LIN {X 0,Y 191.583,Z 536.213,A -85,B 0,C 180,E1 -22027.347,E2 -22027.347} C_VEL
LIN {X 0,Y 188.784,Z 540.752,A -85,B 0,C 180,E1 -22030.427,E2 -22030.427} C_VEL
LIN {X 0,Y 187.171,Z 543.158,A -85,B 0,C 180,E1 -22032.521,E2 -22032.521} C_VEL
LIN {X 0,Y 184.868,Z 546.72,A -85,B 0,C 180,E1 -22036.817,E2 -22036.817} C_VEL
LIN {X 0,Y 184.098,Z 547.887,A -85,B 0,C 180,E1 -22038.998,E2 -22038.998} C_VEL
LIN {X 0,Y 183.22,Z 549.005,A -85,B 0,C 180,E1 -22043.394,E2 -22043.394} C_VEL
LIN {X 0,Y 183.101,Z 548.604,A -85,B 0,C 180,E1 -22047.802,E2 -22047.802} C_VEL
LIN {X 0,Y 183.237,Z 547.778,A -85,B 0,C 180,E1 -22050.002,E2 -22050.002} C_VEL
LIN {X 0,Y 183.088,Z 545.543,A -85,B 0,C 180,E1 -22053.583,E2 -22053.583} C_VEL
LIN {X 0,Y 183.262,Z 542.775,A -85,B 0,C 180,E1 -22056.608,E2 -22056.608} C_VEL
LIN {X 0,Y 183.704,Z 538.696,A -85,B 0,C 180,E1 -22059.915,E2 -22059.915} C_VEL
LIN {X 0,Y 184.708,Z 532.396,A -85,B 0,C 180,E1 -22063.759,E2 -22063.759} C_VEL
LIN {X 0,Y 186.239,Z 525.529,A -85,B 0,C 180,E1 -22067.007,E2 -22067.007} C_VEL
LIN {X 0,Y 187.918,Z 518.509,A -85,B 0,C 180,E1 -22069.671,E2 -22069.671} C_VEL
LIN {X 0,Y 189.702,Z 510.19,A -85,B 0,C 180,E1 -22072.261,E2 -22072.261} C_VEL
LIN {X 0,Y 191.808,Z 500.693,A -85,B 0,C 180,E1 -22074.634,E2 -22074.634} C_VEL
LIN {X 0,Y 194.283,Z 489.109,A -85,B 0,C 180,E1 -22076.885,E2 -22076.885} C_VEL
LIN {X 0,Y 196.502,Z 477.732,A -85,B 0,C 180,E1 -22078.581,E2 -22078.581} C_VEL
LIN {X 0,Y 198.278,Z 466.082,A -85,B 0,C 180,E1 -22079.899,E2 -22079.899} C_VEL
LIN {X 0,Y 199.683,Z 453.556,A -85,B 0,C 180,E1 -22080.908,E2 -22080.908} C_VEL
LIN {X 0,Y 200.634,Z 440.994,A -85,B 0,C 180,E1 -22081.552,E2 -22081.552} C_VEL
LIN {X 0,Y 202.544,Z 391.87,A -85,B 0,C 180,E1 -22083.238,E2 -22083.238} C_VEL
LIN {X 0,Y 200.132,Z 369.782,A -85,B 0,C 180,E1 -22084.491,E2 -22084.491} C_VEL
LIN {X 0,Y 194.209,Z 353.858,A -85,B 0,C 180,E1 -22086.126,E2 -22086.126} C_VEL
LIN {X 0,Y 188.089,Z 340.011,A -85,B 0,C 180,E1 -22087.833,E2 -22087.833} C_VEL
LIN {X 0,Y 186.441,Z 336.416,A -85,B 0,C 180,E1 -22088.331,E2 -22088.331} C_VEL
LIN {X 0,Y 185.481,Z 332.385,A -85,B 0,C 180,E1 -22090.619,E2 -22090.619} C_VEL
LIN {X 0,Y 185.463,Z 332.386,A -85,B 0,C 180,E1 -22096.056,E2 -22096.056} C_VEL
LIN {X 0,Y 185.473,Z 332.384,A -85,B 0,C 180,E1 -22099.896,E2 -22099.896} C_VEL
LIN {X 0,Y 185.512,Z 332.378,A -85,B 0,C 180,E1 -22102.712,E2 -22102.712} C_VEL
LIN {X 0,Y 185.536,Z 332.372,A -85,B 0,C 180,E1 -22107.973,E2 -22107.973} C_VEL
LIN {X 0,Y 185.553,Z 332.371,A -85,B 0,C 180,E1 -22110.596,E2 -22110.596} C_VEL
LIN {X 0,Y 185.586,Z 332.368,A -85,B 0,C 180,E1 -22115.382,E2 -22115.382} C_VEL
LIN {X 0,Y 185.634,Z 332.342,A -85,B 0,C 180,E1 -22121.176,E2 -22121.176} C_VEL
LIN {X 0,Y 185.676,Z 332.354,A -85,B 0,C 180,E1 -22124.635,E2 -22124.635} C_VEL
LIN {X 0,Y 185.894,Z 332.304,A -85,B 0,C 180,E1 -22129.418,E2 -22129.418} C_VEL
LIN {X 0,Y 185.943,Z 332.31,A -85,B 0,C 180,E1 -22133.489,E2 -22133.489} C_VEL
LIN {X 0,Y 186.187,Z 332.289,A -85,B 0,C 180,E1 -22137.836,E2 -22137.836} C_VEL
LIN {X 0,Y 186.402,Z 332.248,A -85,B 0,C 180,E1 -22139.999,E2 -22139.999} C_VEL
LIN {X 0,Y 185.898,Z 332.304,A -85,B 0,C 180,E1 -22144.336,E2 -22144.336} C_VEL
LIN {X 0,Y 185.981,Z 332.318,A -85,B 0,C 180,E1 -22148.693,E2 -22148.693} C_VEL
LIN {X 0,Y 185.724,Z 332.33,A -85,B 0,C 180,E1 -22153.123,E2 -22153.123} C_VEL
LIN {X 0,Y 185.659,Z 332.34,A -85,B 0,C 180,E1 -22157.627,E2 -22157.627} C_VEL
LIN {X 0,Y 185.571,Z 332.367,A -85,B 0,C 180,E1 -22162.254,E2 -22162.254} C_VEL
LIN {X 0,Y 185.582,Z 332.355,A -85,B 0,C 180,E1 -22164.645,E2 -22164.645} C_VEL
LIN {X 0,Y 185.548,Z 332.348,A -85,B 0,C 180,E1 -22169.498,E2 -22169.498} C_VEL
LIN {X 0,Y 185.501,Z 332.372,A -85,B 0,C 180,E1 -22174.631,E2 -22174.631} C_VEL
LIN {X 0,Y 185.508,Z 332.351,A -85,B 0,C 180,E1 -22177.312,E2 -22177.312} C_VEL
LIN {X 0,Y 185.474,Z 332.369,A -85,B 0,C 180,E1 -22180.723,E2 -22180.723} C_VEL
LIN {X 0,Y 185.461,Z 332.368,A -85,B 0,C 180,E1 -22186.054,E2 -22186.054} C_VEL
LIN {X 0,Y 185.47,Z 332.375,A -85,B 0,C 180,E1 -22189.894,E2 -22189.894} C_VEL
LIN {X 0,Y 185.509,Z 332.374,A -85,B 0,C 180,E1 -22192.71,E2 -22192.71} C_VEL
LIN {X 0,Y 185.533,Z 332.374,A -85,B 0,C 180,E1 -22197.971,E2 -22197.971} C_VEL
LIN {X 0,Y 185.549,Z 332.373,A -85,B 0,C 180,E1 -22200.593,E2 -22200.593} C_VEL
LIN {X 0,Y 185.612,Z 332.364,A -85,B 0,C 180,E1 -22205.789,E2 -22205.789} C_VEL
LIN {X 0,Y 186.61,Z 335.177,A -85,B 0,C 180,E1 -22206.126,E2 -22206.126} C_VEL
LIN {X 0,Y 188.138,Z 337.771,A -85,B 0,C 180,E1 -22206.537,E2 -22206.537} C_VEL
LIN {X 0,Y 195.669,Z 351.908,A -85,B 0,C 180,E1 -22208.504,E2 -22208.504} C_VEL
LIN {X 0,Y 199.025,Z 359.752,A -85,B 0,C 180,E1 -22209.387,E2 -22209.387} C_VEL
LIN {X 0,Y 203.412,Z 372.384,A -85,B 0,C 180,E1 -22210.581,E2 -22210.581} C_VEL
LIN {X 0,Y 200.56,Z 435.216,A -85,B 0,C 180,E1 -22212.716,E2 -22212.716} C_VEL
LIN {X 0,Y 199.337,Z 448.756,A -85,B 0,C 180,E1 -22213.562,E2 -22213.562} C_VEL
LIN {X 0,Y 197.947,Z 460.625,A -85,B 0,C 180,E1 -22214.687,E2 -22214.687} C_VEL
LIN {X 0,Y 196.128,Z 472.793,A -85,B 0,C 180,E1 -22216.265,E2 -22216.265} C_VEL
LIN {X 0,Y 193.844,Z 484.802,A -85,B 0,C 180,E1 -22218.321,E2 -22218.321} C_VEL
LIN {X 0,Y 191.638,Z 494.794,A -85,B 0,C 180,E1 -22220.499,E2 -22220.499} C_VEL
LIN {X 0,Y 189.47,Z 504.15,A -85,B 0,C 180,E1 -22223.074,E2 -22223.074} C_VEL
LIN {X 0,Y 187.292,Z 513.207,A -85,B 0,C 180,E1 -22226.233,E2 -22226.233} C_VEL
LIN {X 0,Y 185.605,Z 520.503,A -85,B 0,C 180,E1 -22229.456,E2 -22229.456} C_VEL
LIN {X 0,Y 184.53,Z 525.43,A -85,B 0,C 180,E1 -22232.181,E2 -22232.181} C_VEL
LIN {X 0,Y 183.676,Z 530.659,A -85,B 0,C 180,E1 -22235.83,E2 -22235.83} C_VEL
LIN {X 0,Y 183.13,Z 533.887,A -85,B 0,C 180,E1 -22238.828,E2 -22238.828} C_VEL
LIN {X 0,Y 182.842,Z 535.784,A -85,B 0,C 180,E1 -22241.078,E2 -22241.078} C_VEL
LIN {X 0,Y 182.796,Z 537.198,A -85,B 0,C 180,E1 -22243.335,E2 -22243.335} C_VEL
LIN {X 0,Y 182.939,Z 538.419,A -85,B 0,C 180,E1 -22246.174,E2 -22246.174} C_VEL
LIN {X 0,Y 183.416,Z 538.99,A -85,B 0,C 180,E1 -22250.171,E2 -22250.171} C_VEL
LIN {X 0,Y 184.48,Z 538.359,A -85,B 0,C 180,E1 -22253.893,E2 -22253.893} C_VEL
LIN {X 0,Y 185.784,Z 536.971,A -85,B 0,C 180,E1 -22256.995,E2 -22256.995} C_VEL
LIN {X 0,Y 187.959,Z 534.14,A -85,B 0,C 180,E1 -22260.685,E2 -22260.685} C_VEL
LIN {X 0,Y 191.223,Z 529.402,A -85,B 0,C 180,E1 -22264.725,E2 -22264.725} C_VEL
LIN {X 0,Y 195.104,Z 523.18,A -85,B 0,C 180,E1 -22268.414,E2 -22268.414} C_VEL
LIN {X 0,Y 198.974,Z 516.267,A -85,B 0,C 180,E1 -22271.471,E2 -22271.471} C_VEL
LIN {X 0,Y 202.688,Z 509.169,A -85,B 0,C 180,E1 -22273.903,E2 -22273.903} C_VEL
LIN {X 0,Y 206.691,Z 500.537,A -85,B 0,C 180,E1 -22276.262,E2 -22276.262} C_VEL
LIN {X 0,Y 210.474,Z 491.374,A -85,B 0,C 180,E1 -22278.23,E2 -22278.23} C_VEL
LIN {X 0,Y 214.251,Z 480.505,A -85,B 0,C 180,E1 -22280.061,E2 -22280.061} C_VEL
LIN {X 0,Y 217.541,Z 469.264,A -85,B 0,C 180,E1 -22281.513,E2 -22281.513} C_VEL
LIN {X 0,Y 220.372,Z 457.031,A -85,B 0,C 180,E1 -22282.704,E2 -22282.704} C_VEL
LIN {X 0,Y 222.473,Z 443.681,A -85,B 0,C 180,E1 -22283.632,E2 -22283.632} C_VEL
LIN {X 0,Y 223.846,Z 430.846,A -85,B 0,C 180,E1 -22284.167,E2 -22284.167} C_VEL
LIN {X 0,Y 226.225,Z 394.156,A -85,B 0,C 180,E1 -22285.231,E2 -22285.231} C_VEL
LIN {X 0,Y 220.963,Z 383.068,A -85,B 0,C 180,E1 -22287.269,E2 -22287.269} C_VEL
LIN {X 0,Y 215.515,Z 372.798,A -85,B 0,C 180,E1 -22289.527,E2 -22289.527} C_VEL
LIN {X 0,Y 211.22,Z 365.794,A -85,B 0,C 180,E1 -22291.426,E2 -22291.426} C_VEL
LIN {X 0,Y 205.505,Z 357.753,A -85,B 0,C 180,E1 -22294.149,E2 -22294.149} C_VEL
LIN {X 0,Y 201.846,Z 352.98,A -85,B 0,C 180,E1 -22296.063,E2 -22296.063} C_VEL
LIN {X 0,Y 199.159,Z 349.322,A -85,B 0,C 180,E1 -22297.596,E2 -22297.596} C_VEL
LIN {X 0,Y 195.776,Z 345.444,A -85,B 0,C 180,E1 -22299.658,E2 -22299.658} C_VEL
LIN {X 0,Y 194.816,Z 343.709,A -85,B 0,C 180,E1 -22300.336,E2 -22300.336} C_VEL
LIN {X 0,Y 192.254,Z 341.564,A -85,B 0,C 180,E1 -22302.047,E2 -22302.047} C_VEL
LIN {X 0,Y 190.274,Z 338.16,A -85,B 0,C 180,E1 -22303.642,E2 -22303.642} C_VEL
LIN {X 0,Y 187.582,Z 336.397,A -85,B 0,C 180,E1 -22305.767,E2 -22305.767} C_VEL
LIN {X 0,Y 186.189,Z 334.174,A -85,B 0,C 180,E1 -22307.119,E2 -22307.119} C_VEL
LIN {X 0,Y 185.73,Z 332.335,A -85,B 0,C 180,E1 -22307.78,E2 -22307.78} C_VEL
LIN {X 0,Y 185.963,Z 332.3,A -85,B 0,C 180,E1 -22311.306,E2 -22311.306} C_VEL
LIN {X 0,Y 186.148,Z 332.28,A -85,B 0,C 180,E1 -22317.837,E2 -22317.837} C_VEL
LIN {X 0,Y 186.366,Z 332.267,A -85,B 0,C 180,E1 -22320.001,E2 -22320.001} C_VEL
LIN {X 0,Y 185.873,Z 332.325,A -85,B 0,C 180,E1 -22324.337,E2 -22324.337} C_VEL
LIN {X 0,Y 185.967,Z 332.299,A -85,B 0,C 180,E1 -22328.695,E2 -22328.695} C_VEL
LIN {X 0,Y 185.714,Z 332.328,A -85,B 0,C 180,E1 -22333.125,E2 -22333.125} C_VEL
LIN {X 0,Y 185.677,Z 332.335,A -85,B 0,C 180,E1 -22337.627,E2 -22337.627} C_VEL
LIN {X 0,Y 185.605,Z 332.347,A -85,B 0,C 180,E1 -22343.428,E2 -22343.428} C_VEL
LIN {X 0,Y 185.596,Z 332.595,A -85,B 0,C 180,E1 -22344.664,E2 -22344.664} C_VEL
LIN {X 0,Y 185.914,Z 333.985,A -85,B 0,C 180,E1 -22346.295,E2 -22346.295} C_VEL
LIN {X 0,Y 187.303,Z 336.241,A -85,B 0,C 180,E1 -22347.668,E2 -22347.668} C_VEL
LIN {X 0,Y 191.692,Z 341.119,A -85,B 0,C 180,E1 -22351.222,E2 -22351.222} C_VEL
LIN {X 0,Y 195.213,Z 346.119,A -85,B 0,C 180,E1 -22353.745,E2 -22353.745} C_VEL
LIN {X 0,Y 196.675,Z 348.072,A -85,B 0,C 180,E1 -22354.698,E2 -22354.698} C_VEL
LIN {X 0,Y 200.777,Z 353.997,A -85,B 0,C 180,E1 -22357.174,E2 -22357.174} C_VEL
LIN {X 0,Y 204.53,Z 359.728,A -85,B 0,C 180,E1 -22359.228,E2 -22359.228} C_VEL
LIN {X 0,Y 208.687,Z 366.484,A -85,B 0,C 180,E1 -22361.325,E2 -22361.325} C_VEL
LIN {X 0,Y 213.965,Z 375.728,A -85,B 0,C 180,E1 -22363.769,E2 -22363.769} C_VEL
LIN {X 0,Y 218.853,Z 385.288,A -85,B 0,C 180,E1 -22365.862,E2 -22365.862} C_VEL
LIN {X 0,Y 224.441,Z 397.981,A -85,B 0,C 180,E1 -22368.12,E2 -22368.12} C_VEL
LIN {X 0,Y 225.844,Z 401.455,A -85,B 0,C 180,E1 -22368.668,E2 -22368.668} C_VEL
LIN {X 0,Y 222.983,Z 445.282,A -85,B 0,C 180,E1 -22370.003,E2 -22370.003} C_VEL
LIN {X 0,Y 222.619,Z 448.507,A -85,B 0,C 180,E1 -22370.137,E2 -22370.137} C_VEL
LIN {X 0,Y 221.356,Z 454.274,A -85,B 0,C 180,E1 -22370.283,E2 -22370.283} C_VEL
LIN {X 0,Y 217.615,Z 463.501,A -85,B 0,C 180,E1 -22370.319,E2 -22370.319} C_VEL
LIN {X 0,Y 213.48,Z 472.458,A -85,B 0,C 180,E1 -22370.543,E2 -22370.543} C_VEL
LIN {X 0,Y 211.606,Z 477.79,A -85,B 0,C 180,E1 -22370.988,E2 -22370.988} C_VEL
LIN {X 0,Y 207.869,Z 489.719,A -85,B 0,C 180,E1 -22372.516,E2 -22372.516} C_VEL
LIN {X 0,Y 203.592,Z 500.823,A -85,B 0,C 180,E1 -22374.374,E2 -22374.374} C_VEL
LIN {X 0,Y 199.718,Z 509.796,A -85,B 0,C 180,E1 -22376.344,E2 -22376.344} C_VEL
LIN {X 0,Y 194.763,Z 519.539,A -85,B 0,C 180,E1 -22379.058,E2 -22379.058} C_VEL
LIN {X 0,Y 190.378,Z 527.383,A -85,B 0,C 180,E1 -22381.924,E2 -22381.924} C_VEL
LIN {X 0,Y 186.832,Z 533.565,A -85,B 0,C 180,E1 -22384.897,E2 -22384.897} C_VEL
LIN {X 0,Y 183.033,Z 539.419,A -85,B 0,C 180,E1 -22388.609,E2 -22388.609} C_VEL
LIN {X 0,Y 180.412,Z 543.169,A -85,B 0,C 180,E1 -22391.844,E2 -22391.844} C_VEL
LIN {X 0,Y 178.996,Z 545.117,A -85,B 0,C 180,E1 -22394.05,E2 -22394.05} C_VEL
LIN {X 0,Y 177.945,Z 546.661,A -85,B 0,C 180,E1 -22396.294,E2 -22396.294} C_VEL
LIN {X 0,Y 176.509,Z 548.482,A -85,B 0,C 180,E1 -22400.838,E2 -22400.838} C_VEL
LIN {X 0,Y 176.008,Z 548.783,A -85,B 0,C 180,E1 -22405.422,E2 -22405.422} C_VEL
LIN {X 0,Y 176.019,Z 548.334,A -85,B 0,C 180,E1 -22407.714,E2 -22407.714} C_VEL
LIN {X 0,Y 176.141,Z 547.469,A -85,B 0,C 180,E1 -22410.002,E2 -22410.002} C_VEL
LIN {X 0,Y 175.997,Z 545.487,A -85,B 0,C 180,E1 -22413.321,E2 -22413.321} C_VEL
LIN {X 0,Y 176.205,Z 542.333,A -85,B 0,C 180,E1 -22416.874,E2 -22416.874} C_VEL
LIN {X 0,Y 176.671,Z 538.178,A -85,B 0,C 180,E1 -22420.314,E2 -22420.314} C_VEL
LIN {X 0,Y 177.759,Z 531.795,A -85,B 0,C 180,E1 -22424.308,E2 -22424.308} C_VEL
LIN {X 0,Y 179.431,Z 524.841,A -85,B 0,C 180,E1 -22427.673,E2 -22427.673} C_VEL
LIN {X 0,Y 181.234,Z 517.72,A -85,B 0,C 180,E1 -22430.429,E2 -22430.429} C_VEL
LIN {X 0,Y 183.18,Z 509.067,A -85,B 0,C 180,E1 -22433.159,E2 -22433.159} C_VEL
LIN {X 0,Y 185.676,Z 498.382,A -85,B 0,C 180,E1 -22435.805,E2 -22435.805} C_VEL
LIN {X 0,Y 187.629,Z 489.212,A -85,B 0,C 180,E1 -22437.617,E2 -22437.617} C_VEL
LIN {X 0,Y 189.926,Z 477.908,A -85,B 0,C 180,E1 -22439.362,E2 -22439.362} C_VEL
LIN {X 0,Y 191.766,Z 466.4,A -85,B 0,C 180,E1 -22440.719,E2 -22440.719} C_VEL
LIN {X 0,Y 193.327,Z 453.215,A -85,B 0,C 180,E1 -22441.813,E2 -22441.813} C_VEL
LIN {X 0,Y 194.305,Z 440.553,A -85,B 0,C 180,E1 -22442.475,E2 -22442.475} C_VEL
LIN {X 0,Y 196.253,Z 392.537,A -85,B 0,C 180,E1 -22444.167,E2 -22444.167} C_VEL
LIN {X 0,Y 194.04,Z 371.837,A -85,B 0,C 180,E1 -22445.392,E2 -22445.392} C_VEL
LIN {X 0,Y 187.655,Z 354.77,A -85,B 0,C 180,E1 -22447.26,E2 -22447.26} C_VEL
LIN {X 0,Y 182.372,Z 343.133,A -85,B 0,C 180,E1 -22448.812,E2 -22448.812} C_VEL
LIN {X 0,Y 179.102,Z 336.151,A -85,B 0,C 180,E1 -22449.857,E2 -22449.857} C_VEL
LIN {X 0,Y 178.406,Z 333.266,A -85,B 0,C 180,E1 -22451.695,E2 -22451.695} C_VEL
LIN {X 0,Y 178.397,Z 333.268,A -85,B 0,C 180,E1 -22455.165,E2 -22455.165} C_VEL
LIN {X 0,Y 178.408,Z 333.263,A -85,B 0,C 180,E1 -22458.46,E2 -22458.46} C_VEL
LIN {X 0,Y 178.428,Z 333.26,A -85,B 0,C 180,E1 -22463.784,E2 -22463.784} C_VEL
LIN {X 0,Y 178.489,Z 333.251,A -85,B 0,C 180,E1 -22466.547,E2 -22466.547} C_VEL
LIN {X 0,Y 178.45,Z 333.254,A -85,B 0,C 180,E1 -22471.796,E2 -22471.796} C_VEL
LIN {X 0,Y 178.521,Z 333.247,A -85,B 0,C 180,E1 -22474.889,E2 -22474.889} C_VEL
LIN {X 0,Y 178.563,Z 333.22,A -85,B 0,C 180,E1 -22480.845,E2 -22480.845} C_VEL
LIN {X 0,Y 178.651,Z 333.228,A -85,B 0,C 180,E1 -22486.347,E2 -22486.347} C_VEL
LIN {X 0,Y 178.913,Z 333.167,A -85,B 0,C 180,E1 -22490.959,E2 -22490.959} C_VEL
LIN {X 0,Y 178.849,Z 333.203,A -85,B 0,C 180,E1 -22495.492,E2 -22495.492} C_VEL
LIN {X 0,Y 179.366,Z 333.124,A -85,B 0,C 180,E1 -22499.999,E2 -22499.999} C_VEL
LIN {X 0,Y 178.904,Z 333.194,A -85,B 0,C 180,E1 -22506.768,E2 -22506.768} C_VEL
LIN {X 0,Y 178.838,Z 333.202,A -85,B 0,C 180,E1 -22510.741,E2 -22510.741} C_VEL
LIN {X 0,Y 178.595,Z 333.204,A -85,B 0,C 180,E1 -22515.989,E2 -22515.989} C_VEL
LIN {X 0,Y 178.561,Z 333.234,A -85,B 0,C 180,E1 -22519.153,E2 -22519.153} C_VEL
LIN {X 0,Y 178.52,Z 333.229,A -85,B 0,C 180,E1 -22525.11,E2 -22525.11} C_VEL
LIN {X 0,Y 178.464,Z 333.241,A -85,B 0,C 180,E1 -22530.793,E2 -22530.793} C_VEL
LIN {X 0,Y 178.487,Z 333.245,A -85,B 0,C 180,E1 -22534.217,E2 -22534.217} C_VEL
LIN {X 0,Y 178.398,Z 333.233,A -85,B 0,C 180,E1 -22539.073,E2 -22539.073} C_VEL
LIN {X 0,Y 178.401,Z 333.257,A -85,B 0,C 180,E1 -22542.044,E2 -22542.044} C_VEL
LIN {X 0,Y 178.396,Z 333.255,A -85,B 0,C 180,E1 -22545.163,E2 -22545.163} C_VEL
LIN {X 0,Y 178.405,Z 333.243,A -85,B 0,C 180,E1 -22548.458,E2 -22548.458} C_VEL
LIN {X 0,Y 178.424,Z 333.249,A -85,B 0,C 180,E1 -22553.781,E2 -22553.781} C_VEL
LIN {X 0,Y 178.486,Z 333.243,A -85,B 0,C 180,E1 -22556.544,E2 -22556.544} C_VEL
LIN {X 0,Y 178.446,Z 333.256,A -85,B 0,C 180,E1 -22561.794,E2 -22561.794} C_VEL
LIN {X 0,Y 178.496,Z 333.353,A -85,B 0,C 180,E1 -22564.373,E2 -22564.373} C_VEL
LIN {X 0,Y 179.446,Z 336.032,A -85,B 0,C 180,E1 -22564.706,E2 -22564.706} C_VEL
LIN {X 0,Y 181.005,Z 338.354,A -85,B 0,C 180,E1 -22565.145,E2 -22565.145} C_VEL
LIN {X 0,Y 188.936,Z 353.033,A -85,B 0,C 180,E1 -22567.362,E2 -22567.362} C_VEL
LIN {X 0,Y 192.65,Z 361.062,A -85,B 0,C 180,E1 -22568.375,E2 -22568.375} C_VEL
LIN {X 0,Y 197.1,Z 373.943,A -85,B 0,C 180,E1 -22569.662,E2 -22569.662} C_VEL
LIN {X 0,Y 194.252,Z 434.941,A -85,B 0,C 180,E1 -22571.786,E2 -22571.786} C_VEL
LIN {X 0,Y 193.019,Z 448.221,A -85,B 0,C 180,E1 -22572.62,E2 -22572.62} C_VEL
LIN {X 0,Y 191.58,Z 460.11,A -85,B 0,C 180,E1 -22573.755,E2 -22573.755} C_VEL
LIN {X 0,Y 189.8,Z 471.658,A -85,B 0,C 180,E1 -22575.25,E2 -22575.25} C_VEL
LIN {X 0,Y 187.78,Z 482.209,A -85,B 0,C 180,E1 -22577.021,E2 -22577.021} C_VEL
LIN {X 0,Y 185.382,Z 493.034,A -85,B 0,C 180,E1 -22579.348,E2 -22579.348} C_VEL
LIN {X 0,Y 182.843,Z 503.663,A -85,B 0,C 180,E1 -22582.267,E2 -22582.267} C_VEL
LIN {X 0,Y 180.516,Z 512.847,A -85,B 0,C 180,E1 -22585.532,E2 -22585.532} C_VEL
LIN {X 0,Y 178.709,Z 520.242,A -85,B 0,C 180,E1 -22588.871,E2 -22588.871} C_VEL
LIN {X 0,Y 177.385,Z 526.17,A -85,B 0,C 180,E1 -22592.269,E2 -22592.269} C_VEL
LIN {X 0,Y 176.598,Z 530.93,A -85,B 0,C 180,E1 -22595.786,E2 -22595.786} C_VEL
LIN {X 0,Y 175.968,Z 534.411,A -85,B 0,C 180,E1 -22599.191,E2 -22599.191} C_VEL
LIN {X 0,Y 175.711,Z 536.209,A -85,B 0,C 180,E1 -22601.534,E2 -22601.534} C_VEL
LIN {X 0,Y 175.693,Z 537.573,A -85,B 0,C 180,E1 -22603.885,E2 -22603.885} C_VEL
LIN {X 0,Y 175.85,Z 538.601,A -85,B 0,C 180,E1 -22606.429,E2 -22606.429} C_VEL
LIN {X 0,Y 176.072,Z 539.077,A -85,B 0,C 180,E1 -22608.62,E2 -22608.62} C_VEL
LIN {X 0,Y 176.482,Z 539.171,A -85,B 0,C 180,E1 -22611,E2 -22611} C_VEL
LIN {X 0,Y 177.534,Z 538.59,A -85,B 0,C 180,E1 -22614.427,E2 -22614.427} C_VEL
LIN {X 0,Y 179.164,Z 536.952,A -85,B 0,C 180,E1 -22618.079,E2 -22618.079} C_VEL
LIN {X 0,Y 181.263,Z 534.421,A -85,B 0,C 180,E1 -22621.462,E2 -22621.462} C_VEL
LIN {X 0,Y 184.076,Z 530.632,A -85,B 0,C 180,E1 -22624.936,E2 -22624.936} C_VEL
LIN {X 0,Y 187.649,Z 525.405,A -85,B 0,C 180,E1 -22628.393,E2 -22628.393} C_VEL
LIN {X 0,Y 191.292,Z 519.43,A -85,B 0,C 180,E1 -22631.397,E2 -22631.397} C_VEL
LIN {X 0,Y 195.818,Z 511.415,A -85,B 0,C 180,E1 -22634.47,E2 -22634.47} C_VEL
LIN {X 0,Y 199.885,Z 503.351,A -85,B 0,C 180,E1 -22636.848,E2 -22636.848} C_VEL
LIN {X 0,Y 204.347,Z 493.283,A -85,B 0,C 180,E1 -22639.165,E2 -22639.165} C_VEL
LIN {X 0,Y 208.117,Z 483.339,A -85,B 0,C 180,E1 -22640.956,E2 -22640.956} C_VEL
LIN {X 0,Y 211.591,Z 472.542,A -85,B 0,C 180,E1 -22642.464,E2 -22642.464} C_VEL
LIN {X 0,Y 214.654,Z 460.43,A -85,B 0,C 180,E1 -22643.746,E2 -22643.746} C_VEL
LIN {X 0,Y 217.154,Z 446.95,A -85,B 0,C 180,E1 -22644.777,E2 -22644.777} C_VEL
LIN {X 0,Y 218.683,Z 434.418,A -85,B 0,C 180,E1 -22645.389,E2 -22645.389} C_VEL
LIN {X 0,Y 221.27,Z 396.686,A -85,B 0,C 180,E1 -22646.51,E2 -22646.51} C_VEL
LIN {X 0,Y 215.722,Z 385.017,A -85,B 0,C 180,E1 -22648.81,E2 -22648.81} C_VEL
LIN {X 0,Y 210.131,Z 374.508,A -85,B 0,C 180,E1 -22651.332,E2 -22651.332} C_VEL
LIN {X 0,Y 205.06,Z 366.991,A -85,B 0,C 180,E1 -22653.76,E2 -22653.76} C_VEL
LIN {X 0,Y 202.037,Z 362.773,A -85,B 0,C 180,E1 -22655.328,E2 -22655.328} C_VEL
LIN {X 0,Y 199.351,Z 359.105,A -85,B 0,C 180,E1 -22656.817,E2 -22656.817} C_VEL
LIN {X 0,Y 195.958,Z 354.595,A -85,B 0,C 180,E1 -22658.854,E2 -22658.854} C_VEL
LIN {X 0,Y 193.374,Z 351.4,A -85,B 0,C 180,E1 -22660.546,E2 -22660.546} C_VEL
LIN {X 0,Y 192.535,Z 350.125,A -85,B 0,C 180,E1 -22661.147,E2 -22661.147} C_VEL
LIN {X 0,Y 189.968,Z 347.519,A -85,B 0,C 180,E1 -22662.993,E2 -22662.993} C_VEL
LIN {X 0,Y 188.414,Z 344.857,A -85,B 0,C 180,E1 -22664.311,E2 -22664.311} C_VEL
LIN {X 0,Y 185.69,Z 342.747,A -85,B 0,C 180,E1 -22666.596,E2 -22666.596} C_VEL
LIN {X 0,Y 184.14,Z 339.969,A -85,B 0,C 180,E1 -22668.232,E2 -22668.232} C_VEL
LIN {X 0,Y 183.748,Z 339.136,A -85,B 0,C 180,E1 -22668.696,E2 -22668.696} C_VEL
LIN {X 0,Y 180.696,Z 337.123,A -85,B 0,C 180,E1 -22672.177,E2 -22672.177} C_VEL
LIN {X 0,Y 179.132,Z 334.564,A -85,B 0,C 180,E1 -22674.654,E2 -22674.654} C_VEL
LIN {X 0,Y 178.816,Z 333.195,A -85,B 0,C 180,E1 -22675.492,E2 -22675.492} C_VEL
LIN {X 0,Y 179.331,Z 333.142,A -85,B 0,C 180,E1 -22680.001,E2 -22680.001} C_VEL
LIN {X 0,Y 178.822,Z 333.205,A -85,B 0,C 180,E1 -22684.509,E2 -22684.509} C_VEL
LIN {X 0,Y 178.898,Z 333.182,A -85,B 0,C 180,E1 -22689.041,E2 -22689.041} C_VEL
LIN {X 0,Y 178.642,Z 333.209,A -85,B 0,C 180,E1 -22693.654,E2 -22693.654} C_VEL
LIN {X 0,Y 178.653,Z 333.346,A -85,B 0,C 180,E1 -22698.047,E2 -22698.047} C_VEL
LIN {X 0,Y 179.263,Z 335.526,A -85,B 0,C 180,E1 -22699.371,E2 -22699.371} C_VEL
LIN {X 0,Y 181,Z 337.81,A -85,B 0,C 180,E1 -22701.946,E2 -22701.946} C_VEL
LIN {X 0,Y 183.17,Z 339.266,A -85,B 0,C 180,E1 -22704.434,E2 -22704.434} C_VEL
LIN {X 0,Y 184.264,Z 340.742,A -85,B 0,C 180,E1 -22705.637,E2 -22705.637} C_VEL
LIN {X 0,Y 186.143,Z 343.345,A -85,B 0,C 180,E1 -22707.498,E2 -22707.498} C_VEL
LIN {X 0,Y 189.689,Z 347.557,A -85,B 0,C 180,E1 -22710.492,E2 -22710.492} C_VEL
LIN {X 0,Y 193.668,Z 353.099,A -85,B 0,C 180,E1 -22713.425,E2 -22713.425} C_VEL
LIN {X 0,Y 198.443,Z 360.395,A -85,B 0,C 180,E1 -22716.499,E2 -22716.499} C_VEL
LIN {X 0,Y 202.066,Z 366.095,A -85,B 0,C 180,E1 -22718.567,E2 -22718.567} C_VEL
LIN {X 0,Y 206.868,Z 374.136,A -85,B 0,C 180,E1 -22721.069,E2 -22721.069} C_VEL
LIN {X 0,Y 212.769,Z 385.172,A -85,B 0,C 180,E1 -22723.87,E2 -22723.87} C_VEL
LIN {X 0,Y 218.144,Z 397.116,A -85,B 0,C 180,E1 -22726.24,E2 -22726.24} C_VEL
LIN {X 0,Y 220.886,Z 403.815,A -85,B 0,C 180,E1 -22727.388,E2 -22727.388} C_VEL
LIN {X 0,Y 218.081,Z 445.079,A -85,B 0,C 180,E1 -22728.662,E2 -22728.662} C_VEL
LIN {X 0,Y 216.179,Z 458.675,A -85,B 0,C 180,E1 -22729.385,E2 -22729.385} C_VEL
LIN {X 0,Y 213.371,Z 471.362,A -85,B 0,C 180,E1 -22730.347,E2 -22730.347} C_VEL
LIN {X 0,Y 211.606,Z 477.79,A -85,B 0,C 180,E1 -22730.988,E2 -22730.988} C_VEL
LIN {X 0,Y 209.565,Z 483.147,A -85,B 0,C 180,E1 -22731.497,E2 -22731.497} C_VEL
LIN {X 0,Y 204.49,Z 491.501,A -85,B 0,C 180,E1 -22732.082,E2 -22732.082} C_VEL
LIN {X 0,Y 199.21,Z 499.342,A -85,B 0,C 180,E1 -22732.861,E2 -22732.861} C_VEL
LIN {X 0,Y 196.854,Z 503.881,A -85,B 0,C 180,E1 -22733.675,E2 -22733.675} C_VEL
LIN {X 0,Y 192.104,Z 513.776,A -85,B 0,C 180,E1 -22736.091,E2 -22736.091} C_VEL
LIN {X 0,Y 187.15,Z 522.68,A -85,B 0,C 180,E1 -22738.915,E2 -22738.915} C_VEL
LIN {X 0,Y 182.786,Z 529.87,A -85,B 0,C 180,E1 -22741.903,E2 -22741.903} C_VEL
LIN {X 0,Y 179.735,Z 534.741,A -85,B 0,C 180,E1 -22744.527,E2 -22744.527} C_VEL
LIN {X 0,Y 176.425,Z 539.504,A -85,B 0,C 180,E1 -22747.765,E2 -22747.765} C_VEL
LIN {X 0,Y 173.68,Z 543.18,A -85,B 0,C 180,E1 -22751.114,E2 -22751.114} C_VEL
LIN {X 0,Y 172.152,Z 545.094,A -85,B 0,C 180,E1 -22753.397,E2 -22753.397} C_VEL
LIN {X 0,Y 171.024,Z 546.583,A -85,B 0,C 180,E1 -22755.728,E2 -22755.728} C_VEL
LIN {X 0,Y 169.488,Z 548.33,A -85,B 0,C 180,E1 -22760.455,E2 -22760.455} C_VEL
LIN {X 0,Y 168.931,Z 548.56,A -85,B 0,C 180,E1 -22765.229,E2 -22765.229} C_VEL
LIN {X 0,Y 168.948,Z 548.057,A -85,B 0,C 180,E1 -22767.618,E2 -22767.618} C_VEL
LIN {X 0,Y 169.047,Z 547.159,A -85,B 0,C 180,E1 -22770.002,E2 -22770.002} C_VEL
LIN {X 0,Y 168.904,Z 545.46,A -85,B 0,C 180,E1 -22772.994,E2 -22772.994} C_VEL
LIN {X 0,Y 169.141,Z 541.887,A -85,B 0,C 180,E1 -22777.163,E2 -22777.163} C_VEL
LIN {X 0,Y 169.661,Z 537.658,A -85,B 0,C 180,E1 -22780.745,E2 -22780.745} C_VEL
LIN {X 0,Y 170.851,Z 531.194,A -85,B 0,C 180,E1 -22784.9,E2 -22784.9} C_VEL
LIN {X 0,Y 172.641,Z 524.131,A -85,B 0,C 180,E1 -22788.393,E2 -22788.393} C_VEL
LIN {X 0,Y 174.842,Z 515.736,A -85,B 0,C 180,E1 -22791.648,E2 -22791.648} C_VEL
LIN {X 0,Y 176.131,Z 509.994,A -85,B 0,C 180,E1 -22793.519,E2 -22793.519} C_VEL
LIN {X 0,Y 178.683,Z 499.618,A -85,B 0,C 180,E1 -22796.265,E2 -22796.265} C_VEL
LIN {X 0,Y 181.009,Z 489.316,A -85,B 0,C 180,E1 -22798.402,E2 -22798.402} C_VEL
LIN {X 0,Y 183.39,Z 478.084,A -85,B 0,C 180,E1 -22800.2,E2 -22800.2} C_VEL
LIN {X 0,Y 185.474,Z 465.474,A -85,B 0,C 180,E1 -22801.721,E2 -22801.721} C_VEL
LIN {X 0,Y 187.023,Z 452.874,A -85,B 0,C 180,E1 -22802.778,E2 -22802.778} C_VEL
LIN {X 0,Y 188.026,Z 440.111,A -85,B 0,C 180,E1 -22803.46,E2 -22803.46} C_VEL
LIN {X 0,Y 190.014,Z 393.317,A -85,B 0,C 180,E1 -22805.154,E2 -22805.154} C_VEL
LIN {X 0,Y 188.013,Z 374.013,A -85,B 0,C 180,E1 -22806.344,E2 -22806.344} C_VEL
LIN {X 0,Y 182.154,Z 358.233,A -85,B 0,C 180,E1 -22808.157,E2 -22808.157} C_VEL
LIN {X 0,Y 177.148,Z 346.991,A -85,B 0,C 180,E1 -22809.722,E2 -22809.722} C_VEL
LIN {X 0,Y 172.926,Z 338.597,A -85,B 0,C 180,E1 -22811.082,E2 -22811.082} C_VEL
LIN {X 0,Y 171.798,Z 335.894,A -85,B 0,C 180,E1 -22811.528,E2 -22811.528} C_VEL
LIN {X 0,Y 171.334,Z 334.148,A -85,B 0,C 180,E1 -22812.712,E2 -22812.712} C_VEL
LIN {X 0,Y 171.34,Z 334.147,A -85,B 0,C 180,E1 -22817.591,E2 -22817.591} C_VEL
LIN {X 0,Y 171.392,Z 334.133,A -85,B 0,C 180,E1 -22822.042,E2 -22822.042} C_VEL
LIN {X 0,Y 171.403,Z 334.131,A -85,B 0,C 180,E1 -22825.093,E2 -22825.093} C_VEL
LIN {X 0,Y 171.414,Z 334.132,A -85,B 0,C 180,E1 -22830.527,E2 -22830.527} C_VEL
LIN {X 0,Y 171.446,Z 334.128,A -85,B 0,C 180,E1 -22835.799,E2 -22835.799} C_VEL
LIN {X 0,Y 171.517,Z 334.096,A -85,B 0,C 180,E1 -22840.864,E2 -22840.864} C_VEL
LIN {X 0,Y 171.566,Z 334.112,A -85,B 0,C 180,E1 -22845.771,E2 -22845.771} C_VEL
LIN {X 0,Y 171.851,Z 334.045,A -85,B 0,C 180,E1 -22850.584,E2 -22850.584} C_VEL
LIN {X 0,Y 171.799,Z 334.08,A -85,B 0,C 180,E1 -22855.306,E2 -22855.306} C_VEL
LIN {X 0,Y 172.329,Z 333.999,A -85,B 0,C 180,E1 -22859.999,E2 -22859.999} C_VEL
LIN {X 0,Y 171.867,Z 334.073,A -85,B 0,C 180,E1 -22867.046,E2 -22867.046} C_VEL
LIN {X 0,Y 171.773,Z 334.081,A -85,B 0,C 180,E1 -22870.894,E2 -22870.894} C_VEL
LIN {X 0,Y 171.525,Z 334.088,A -85,B 0,C 180,E1 -22876.667,E2 -22876.667} C_VEL
LIN {X 0,Y 171.436,Z 334.128,A -85,B 0,C 180,E1 -22881.651,E2 -22881.651} C_VEL
LIN {X 0,Y 171.447,Z 334.106,A -85,B 0,C 180,E1 -22885.597,E2 -22885.597} C_VEL
LIN {X 0,Y 171.421,Z 334.118,A -85,B 0,C 180,E1 -22890.571,E2 -22890.571} C_VEL
LIN {X 0,Y 171.396,Z 334.126,A -85,B 0,C 180,E1 -22895.033,E2 -22895.033} C_VEL
LIN {X 0,Y 171.352,Z 334.109,A -85,B 0,C 180,E1 -22898.802,E2 -22898.802} C_VEL
LIN {X 0,Y 171.324,Z 334.14,A -85,B 0,C 180,E1 -22904.216,E2 -22904.216} C_VEL
LIN {X 0,Y 171.338,Z 334.126,A -85,B 0,C 180,E1 -22908.98,E2 -22908.98} C_VEL
LIN {X 0,Y 171.389,Z 334.136,A -85,B 0,C 180,E1 -22912.039,E2 -22912.039} C_VEL
LIN {X 0,Y 171.4,Z 334.118,A -85,B 0,C 180,E1 -22915.091,E2 -22915.091} C_VEL
LIN {X 0,Y 171.411,Z 334.135,A -85,B 0,C 180,E1 -22920.525,E2 -22920.525} C_VEL
LIN {X 0,Y 171.384,Z 334.138,A -85,B 0,C 180,E1 -22922.773,E2 -22922.773} C_VEL
LIN {X 0,Y 172.439,Z 337.039,A -85,B 0,C 180,E1 -22923.191,E2 -22923.191} C_VEL
LIN {X 0,Y 174.118,Z 339.587,A -85,B 0,C 180,E1 -22923.705,E2 -22923.705} C_VEL
LIN {X 0,Y 179.245,Z 348.487,A -85,B 0,C 180,E1 -22925.258,E2 -22925.258} C_VEL
LIN {X 0,Y 186.209,Z 362.201,A -85,B 0,C 180,E1 -22927.266,E2 -22927.266} C_VEL
LIN {X 0,Y 190.847,Z 375.458,A -85,B 0,C 180,E1 -22928.682,E2 -22928.682} C_VEL
LIN {X 0,Y 187.924,Z 435.346,A -85,B 0,C 180,E1 -22930.826,E2 -22930.826} C_VEL
LIN {X 0,Y 186.645,Z 448.601,A -85,B 0,C 180,E1 -22931.687,E2 -22931.687} C_VEL
LIN {X 0,Y 185.099,Z 460.726,A -85,B 0,C 180,E1 -22932.885,E2 -22932.885} C_VEL
LIN {X 0,Y 183.253,Z 472.173,A -85,B 0,C 180,E1 -22934.425,E2 -22934.425} C_VEL
LIN {X 0,Y 181.112,Z 482.762,A -85,B 0,C 180,E1 -22936.273,E2 -22936.273} C_VEL
LIN {X 0,Y 178.647,Z 493.431,A -85,B 0,C 180,E1 -22938.654,E2 -22938.654} C_VEL
LIN {X 0,Y 176.248,Z 503.131,A -85,B 0,C 180,E1 -22941.398,E2 -22941.398} C_VEL
LIN {X 0,Y 174.118,Z 511.092,A -85,B 0,C 180,E1 -22944.206,E2 -22944.206} C_VEL
LIN {X 0,Y 172.096,Z 518.857,A -85,B 0,C 180,E1 -22947.657,E2 -22947.657} C_VEL
LIN {X 0,Y 170.642,Z 525.077,A -85,B 0,C 180,E1 -22951.178,E2 -22951.178} C_VEL
LIN {X 0,Y 169.697,Z 530.017,A -85,B 0,C 180,E1 -22954.749,E2 -22954.749} C_VEL
LIN {X 0,Y 168.984,Z 533.842,A -85,B 0,C 180,E1 -22958.368,E2 -22958.368} C_VEL
LIN {X 0,Y 168.584,Z 536.633,A -85,B 0,C 180,E1 -22962.029,E2 -22962.029} C_VEL
LIN {X 0,Y 168.786,Z 538.789,A -85,B 0,C 180,E1 -22966.729,E2 -22966.729} C_VEL
LIN {X 0,Y 169.096,Z 539.306,A -85,B 0,C 180,E1 -22969.418,E2 -22969.418} C_VEL
LIN {X 0,Y 169.597,Z 539.352,A -85,B 0,C 180,E1 -22971.895,E2 -22971.895} C_VEL
LIN {X 0,Y 170.627,Z 538.815,A -85,B 0,C 180,E1 -22975.021,E2 -22975.021} C_VEL
LIN {X 0,Y 172.609,Z 536.933,A -85,B 0,C 180,E1 -22979.246,E2 -22979.246} C_VEL
LIN {X 0,Y 174.623,Z 534.695,A -85,B 0,C 180,E1 -22982.309,E2 -22982.309} C_VEL
LIN {X 0,Y 178.007,Z 530.401,A -85,B 0,C 180,E1 -22986.312,E2 -22986.312} C_VEL
LIN {X 0,Y 181.617,Z 525.414,A -85,B 0,C 180,E1 -22989.643,E2 -22989.643} C_VEL
LIN {X 0,Y 185.777,Z 518.958,A -85,B 0,C 180,E1 -22992.914,E2 -22992.914} C_VEL
LIN {X 0,Y 189.597,Z 512.48,A -85,B 0,C 180,E1 -22995.446,E2 -22995.446} C_VEL
LIN {X 0,Y 193.994,Z 504.321,A -85,B 0,C 180,E1 -22997.956,E2 -22997.956} C_VEL
LIN {X 0,Y 198.601,Z 494.455,A -85,B 0,C 180,E1 -23000.307,E2 -23000.307} C_VEL
LIN {X 0,Y 203.029,Z 483.321,A -85,B 0,C 180,E1 -23002.354,E2 -23002.354} C_VEL
LIN {X 0,Y 206.647,Z 472.455,A -85,B 0,C 180,E1 -23003.871,E2 -23003.871} C_VEL
LIN {X 0,Y 209.777,Z 460.503,A -85,B 0,C 180,E1 -23005.137,E2 -23005.137} C_VEL
LIN {X 0,Y 212.241,Z 447.678,A -85,B 0,C 180,E1 -23006.132,E2 -23006.132} C_VEL
LIN {X 0,Y 213.829,Z 435.499,A -85,B 0,C 180,E1 -23006.754,E2 -23006.754} C_VEL
LIN {X 0,Y 216.423,Z 399.326,A -85,B 0,C 180,E1 -23007.844,E2 -23007.844} C_VEL
LIN {X 0,Y 210.816,Z 387.285,A -85,B 0,C 180,E1 -23010.362,E2 -23010.362} C_VEL
LIN {X 0,Y 205.722,Z 377.961,A -85,B 0,C 180,E1 -23012.82,E2 -23012.82} C_VEL
LIN {X 0,Y 199.849,Z 369.316,A -85,B 0,C 180,E1 -23015.886,E2 -23015.886} C_VEL
LIN {X 0,Y 196.577,Z 364.822,A -85,B 0,C 180,E1 -23017.777,E2 -23017.777} C_VEL
LIN {X 0,Y 193.753,Z 360.944,A -85,B 0,C 180,E1 -23019.567,E2 -23019.567} C_VEL
LIN {X 0,Y 191.024,Z 357.366,A -85,B 0,C 180,E1 -23021.454,E2 -23021.454} C_VEL
LIN {X 0,Y 189.87,Z 356.054,A -85,B 0,C 180,E1 -23022.295,E2 -23022.295} C_VEL
LIN {X 0,Y 187.302,Z 352.757,A -85,B 0,C 180,E1 -23024.346,E2 -23024.346} C_VEL
LIN {X 0,Y 186.548,Z 351.474,A -85,B 0,C 180,E1 -23025.024,E2 -23025.024} C_VEL
LIN {X 0,Y 183.76,Z 348.964,A -85,B 0,C 180,E1 -23027.525,E2 -23027.525} C_VEL
LIN {X 0,Y 182.116,Z 345.913,A -85,B 0,C 180,E1 -23029.403,E2 -23029.403} C_VEL
LIN {X 0,Y 179.111,Z 343.576,A -85,B 0,C 180,E1 -23033.099,E2 -23033.099} C_VEL
LIN {X 0,Y 177.63,Z 340.668,A -85,B 0,C 180,E1 -23035.746,E2 -23035.746} C_VEL
LIN {X 0,Y 177.517,Z 340.197,A -85,B 0,C 180,E1 -23036.028,E2 -23036.028} C_VEL
LIN {X 0,Y 174.983,Z 338.941,A -85,B 0,C 180,E1 -23042.302,E2 -23042.302} C_VEL
LIN {X 0,Y 174.587,Z 338.841,A -85,B 0,C 180,E1 -23049.267,E2 -23049.267} C_VEL
LIN {X 0,Y 177.375,Z 340.386,A -85,B 0,C 180,E1 -23057.437,E2 -23057.437} C_VEL
LIN {X 0,Y 178.509,Z 343.251,A -85,B 0,C 180,E1 -23059.709,E2 -23059.709} C_VEL
LIN {X 0,Y 180.834,Z 345.42,A -85,B 0,C 180,E1 -23062.871,E2 -23062.871} C_VEL
LIN {X 0,Y 182.181,Z 346.476,A -85,B 0,C 180,E1 -23064.398,E2 -23064.398} C_VEL
LIN {X 0,Y 184.375,Z 349.844,A -85,B 0,C 180,E1 -23066.761,E2 -23066.761} C_VEL
LIN {X 0,Y 187.829,Z 354.156,A -85,B 0,C 180,E1 -23069.83,E2 -23069.83} C_VEL
LIN {X 0,Y 192.062,Z 360.417,A -85,B 0,C 180,E1 -23073.089,E2 -23073.089} C_VEL
LIN {X 0,Y 195.946,Z 366.434,A -85,B 0,C 180,E1 -23075.684,E2 -23075.684} C_VEL
LIN {X 0,Y 199.953,Z 373.016,A -85,B 0,C 180,E1 -23078.075,E2 -23078.075} C_VEL
LIN {X 0,Y 204.381,Z 380.809,A -85,B 0,C 180,E1 -23080.478,E2 -23080.478} C_VEL
LIN {X 0,Y 209.381,Z 390.511,A -85,B 0,C 180,E1 -23082.969,E2 -23082.969} C_VEL
LIN {X 0,Y 214.53,Z 402.373,A -85,B 0,C 180,E1 -23085.376,E2 -23085.376} C_VEL
LIN {X 0,Y 216.018,Z 406.126,A -85,B 0,C 180,E1 -23086.04,E2 -23086.04} C_VEL
LIN {X 0,Y 213.308,Z 444.839,A -85,B 0,C 180,E1 -23087.259,E2 -23087.259} C_VEL
LIN {X 0,Y 211.41,Z 458.158,A -85,B 0,C 180,E1 -23087.973,E2 -23087.973} C_VEL
LIN {X 0,Y 208.491,Z 470.805,A -85,B 0,C 180,E1 -23088.907,E2 -23088.907} C_VEL
LIN {X 0,Y 204.848,Z 483.349,A -85,B 0,C 180,E1 -23090.286,E2 -23090.286} C_VEL
LIN {X 0,Y 200.871,Z 494.533,A -85,B 0,C 180,E1 -23091.93,E2 -23091.93} C_VEL
LIN {X 0,Y 196.854,Z 503.881,A -85,B 0,C 180,E1 -23093.675,E2 -23093.675} C_VEL
LIN {X 0,Y 194.45,Z 508.306,A -85,B 0,C 180,E1 -23094.576,E2 -23094.576} C_VEL
LIN {X 0,Y 188.702,Z 515.184,A -85,B 0,C 180,E1 -23095.849,E2 -23095.849} C_VEL
LIN {X 0,Y 182.663,Z 521.491,A -85,B 0,C 180,E1 -23097.323,E2 -23097.323} C_VEL
LIN {X 0,Y 179.867,Z 525.012,A -85,B 0,C 180,E1 -23098.539,E2 -23098.539} C_VEL
LIN {X 0,Y 175.877,Z 531.122,A -85,B 0,C 180,E1 -23101.349,E2 -23101.349} C_VEL
LIN {X 0,Y 172.118,Z 536.59,A -85,B 0,C 180,E1 -23104.615,E2 -23104.615} C_VEL
LIN {X 0,Y 168.849,Z 540.903,A -85,B 0,C 180,E1 -23108.003,E2 -23108.003} C_VEL
LIN {X 0,Y 166.951,Z 543.198,A -85,B 0,C 180,E1 -23110.322,E2 -23110.322} C_VEL
LIN {X 0,Y 165.334,Z 545.073,A -85,B 0,C 180,E1 -23112.692,E2 -23112.692} C_VEL
LIN {X 0,Y 163.166,Z 547.527,A -85,B 0,C 180,E1 -23117.566,E2 -23117.566} C_VEL
LIN {X 0,Y 162.032,Z 548.454,A -85,B 0,C 180,E1 -23122.526,E2 -23122.526} C_VEL
LIN {X 0,Y 161.834,Z 547.864,A -85,B 0,C 180,E1 -23127.234,E2 -23127.234} C_VEL
LIN {X 0,Y 161.956,Z 546.849,A -85,B 0,C 180,E1 -23130.002,E2 -23130.002} C_VEL
LIN {X 0,Y 161.835,Z 545.335,A -85,B 0,C 180,E1 -23132.771,E2 -23132.771} C_VEL
LIN {X 0,Y 161.973,Z 542.639,A -85,B 0,C 180,E1 -23136.23,E2 -23136.23} C_VEL
LIN {X 0,Y 162.395,Z 538.711,A -85,B 0,C 180,E1 -23139.971,E2 -23139.971} C_VEL
LIN {X 0,Y 163.477,Z 532.634,A -85,B 0,C 180,E1 -23144.314,E2 -23144.314} C_VEL
LIN {X 0,Y 165.165,Z 525.953,A -85,B 0,C 180,E1 -23147.971,E2 -23147.971} C_VEL
LIN {X 0,Y 166.995,Z 519.138,A -85,B 0,C 180,E1 -23150.963,E2 -23150.963} C_VEL
LIN {X 0,Y 168.174,Z 514.645,A -85,B 0,C 180,E1 -23152.643,E2 -23152.643} C_VEL
LIN {X 0,Y 170.638,Z 505.129,A -85,B 0,C 180,E1 -23155.626,E2 -23155.626} C_VEL
LIN {X 0,Y 173.148,Z 494.809,A -85,B 0,C 180,E1 -23158.157,E2 -23158.157} C_VEL
LIN {X 0,Y 175.844,Z 483.378,A -85,B 0,C 180,E1 -23160.306,E2 -23160.306} C_VEL
LIN {X 0,Y 178.115,Z 471.461,A -85,B 0,C 180,E1 -23162.022,E2 -23162.022} C_VEL
LIN {X 0,Y 179.941,Z 459.034,A -85,B 0,C 180,E1 -23163.317,E2 -23163.317} C_VEL
LIN {X 0,Y 181.306,Z 446.366,A -85,B 0,C 180,E1 -23164.201,E2 -23164.201} C_VEL
LIN {X 0,Y 182.553,Z 423.663,A -85,B 0,C 180,E1 -23165.107,E2 -23165.107} C_VEL
LIN {X 0,Y 183.831,Z 393.958,A -85,B 0,C 180,E1 -23166.211,E2 -23166.211} C_VEL
LIN {X 0,Y 182.039,Z 376.24,A -85,B 0,C 180,E1 -23167.349,E2 -23167.349} C_VEL
LIN {X 0,Y 176.461,Z 361.064,A -85,B 0,C 180,E1 -23169.189,E2 -23169.189} C_VEL
LIN {X 0,Y 170.761,Z 348.181,A -85,B 0,C 180,E1 -23171.103,E2 -23171.103} C_VEL
LIN {X 0,Y 166.031,Z 339.117,A -85,B 0,C 180,E1 -23172.731,E2 -23172.731} C_VEL
LIN {X 0,Y 164.385,Z 335.677,A -85,B 0,C 180,E1 -23173.38,E2 -23173.38} C_VEL
LIN {X 0,Y 164.294,Z 335.024,A -85,B 0,C 180,E1 -23173.954,E2 -23173.954} C_VEL
LIN {X 0,Y 164.268,Z 335.028,A -85,B 0,C 180,E1 -23176.8,E2 -23176.8} C_VEL
LIN {X 0,Y 164.301,Z 335.022,A -85,B 0,C 180,E1 -23180.353,E2 -23180.353} C_VEL
LIN {X 0,Y 164.336,Z 335.013,A -85,B 0,C 180,E1 -23184.35,E2 -23184.35} C_VEL
LIN {X 0,Y 164.376,Z 335.006,A -85,B 0,C 180,E1 -23189.131,E2 -23189.131} C_VEL
LIN {X 0,Y 164.4,Z 335.006,A -85,B 0,C 180,E1 -23194.691,E2 -23194.691} C_VEL
LIN {X 0,Y 164.423,Z 334.977,A -85,B 0,C 180,E1 -23200.116,E2 -23200.116} C_VEL
LIN {X 0,Y 164.493,Z 334.995,A -85,B 0,C 180,E1 -23205.146,E2 -23205.146} C_VEL
LIN {X 0,Y 164.771,Z 334.926,A -85,B 0,C 180,E1 -23210.176,E2 -23210.176} C_VEL
LIN {X 0,Y 164.83,Z 334.93,A -85,B 0,C 180,E1 -23212.65,E2 -23212.65} C_VEL
LIN {X 0,Y 165.291,Z 334.875,A -85,B 0,C 180,E1 -23219.999,E2 -23219.999} C_VEL
LIN {X 0,Y 164.828,Z 334.949,A -85,B 0,C 180,E1 -23227.349,E2 -23227.349} C_VEL
LIN {X 0,Y 164.707,Z 334.96,A -85,B 0,C 180,E1 -23231.058,E2 -23231.058} C_VEL
LIN {X 0,Y 164.444,Z 334.975,A -85,B 0,C 180,E1 -23237.407,E2 -23237.407} C_VEL
LIN {X 0,Y 164.361,Z 335.009,A -85,B 0,C 180,E1 -23242.633,E2 -23242.633} C_VEL
LIN {X 0,Y 164.374,Z 334.979,A -85,B 0,C 180,E1 -23246.115,E2 -23246.115} C_VEL
LIN {X 0,Y 164.361,Z 334.999,A -85,B 0,C 180,E1 -23251.216,E2 -23251.216} C_VEL
LIN {X 0,Y 164.286,Z 334.995,A -85,B 0,C 180,E1 -23256.791,E2 -23256.791} C_VEL
LIN {X 0,Y 164.292,Z 334.994,A -85,B 0,C 180,E1 -23259.915,E2 -23259.915} C_VEL
LIN {X 0,Y 164.283,Z 335.019,A -85,B 0,C 180,E1 -23263.34,E2 -23263.34} C_VEL
LIN {X 0,Y 164.266,Z 335.001,A -85,B 0,C 180,E1 -23266.797,E2 -23266.797} C_VEL
LIN {X 0,Y 164.298,Z 335.015,A -85,B 0,C 180,E1 -23270.35,E2 -23270.35} C_VEL
LIN {X 0,Y 164.332,Z 334.999,A -85,B 0,C 180,E1 -23274.347,E2 -23274.347} C_VEL
LIN {X 0,Y 164.374,Z 335.01,A -85,B 0,C 180,E1 -23280.334,E2 -23280.334} C_VEL
LIN {X 0,Y 164.371,Z 335.01,A -85,B 0,C 180,E1 -23281.073,E2 -23281.073} C_VEL
LIN {X 0,Y 165.36,Z 337.834,A -85,B 0,C 180,E1 -23281.489,E2 -23281.489} C_VEL
LIN {X 0,Y 166.904,Z 340.073,A -85,B 0,C 180,E1 -23282.003,E2 -23282.003} C_VEL
LIN {X 0,Y 173.774,Z 351.856,A -85,B 0,C 180,E1 -23284.238,E2 -23284.238} C_VEL
LIN {X 0,Y 180.694,Z 365.552,A -85,B 0,C 180,E1 -23286.358,E2 -23286.358} C_VEL
LIN {X 0,Y 184.719,Z 377.429,A -85,B 0,C 180,E1 -23287.673,E2 -23287.673} C_VEL
LIN {X 0,Y 181.598,Z 436.33,A -85,B 0,C 180,E1 -23289.836,E2 -23289.836} C_VEL
LIN {X 0,Y 180.201,Z 450.076,A -85,B 0,C 180,E1 -23290.786,E2 -23290.786} C_VEL
LIN {X 0,Y 178.492,Z 462.416,A -85,B 0,C 180,E1 -23292.083,E2 -23292.083} C_VEL
LIN {X 0,Y 176.45,Z 474.245,A -85,B 0,C 180,E1 -23293.809,E2 -23293.809} C_VEL
LIN {X 0,Y 173.988,Z 485.656,A -85,B 0,C 180,E1 -23295.972,E2 -23295.972} C_VEL
LIN {X 0,Y 171.388,Z 495.961,A -85,B 0,C 180,E1 -23298.466,E2 -23298.466} C_VEL
LIN {X 0,Y 169.192,Z 504.367,A -85,B 0,C 180,E1 -23301.036,E2 -23301.036} C_VEL
LIN {X 0,Y 166.669,Z 513.491,A -85,B 0,C 180,E1 -23304.554,E2 -23304.554} C_VEL
LIN {X 0,Y 164.692,Z 520.846,A -85,B 0,C 180,E1 -23308.164,E2 -23308.164} C_VEL
LIN {X 0,Y 163.49,Z 525.817,A -85,B 0,C 180,E1 -23311.229,E2 -23311.229} C_VEL
LIN {X 0,Y 162.541,Z 530.644,A -85,B 0,C 180,E1 -23314.959,E2 -23314.959} C_VEL
LIN {X 0,Y 161.822,Z 534.366,A -85,B 0,C 180,E1 -23318.741,E2 -23318.741} C_VEL
LIN {X 0,Y 161.472,Z 537.056,A -85,B 0,C 180,E1 -23322.567,E2 -23322.567} C_VEL
LIN {X 0,Y 161.709,Z 538.97,A -85,B 0,C 180,E1 -23327.035,E2 -23327.035} C_VEL
LIN {X 0,Y 162.137,Z 539.537,A -85,B 0,C 180,E1 -23330.287,E2 -23330.287} C_VEL
LIN {X 0,Y 162.743,Z 539.534,A -85,B 0,C 180,E1 -23332.869,E2 -23332.869} C_VEL
LIN {X 0,Y 163.735,Z 539.043,A -85,B 0,C 180,E1 -23335.661,E2 -23335.661} C_VEL
LIN {X 0,Y 166.139,Z 536.919,A -85,B 0,C 180,E1 -23340.503,E2 -23340.503} C_VEL
LIN {X 0,Y 168.693,Z 534.209,A -85,B 0,C 180,E1 -23344.077,E2 -23344.077} C_VEL
LIN {X 0,Y 172.058,Z 530.174,A -85,B 0,C 180,E1 -23347.782,E2 -23347.782} C_VEL
LIN {X 0,Y 175.962,Z 525.026,A -85,B 0,C 180,E1 -23351.22,E2 -23351.22} C_VEL
LIN {X 0,Y 180.364,Z 518.447,A -85,B 0,C 180,E1 -23354.535,E2 -23354.535} C_VEL
LIN {X 0,Y 185.472,Z 510.148,A -85,B 0,C 180,E1 -23357.635,E2 -23357.635} C_VEL
LIN {X 0,Y 190.044,Z 501.599,A -85,B 0,C 180,E1 -23360.113,E2 -23360.113} C_VEL
LIN {X 0,Y 194.455,Z 492.269,A -85,B 0,C 180,E1 -23362.216,E2 -23362.216} C_VEL
LIN {X 0,Y 198.573,Z 481.863,A -85,B 0,C 180,E1 -23364.053,E2 -23364.053} C_VEL
LIN {X 0,Y 202.355,Z 470.53,A -85,B 0,C 180,E1 -23365.571,E2 -23365.571} C_VEL
LIN {X 0,Y 205.716,Z 457.622,A -85,B 0,C 180,E1 -23366.865,E2 -23366.865} C_VEL
LIN {X 0,Y 208.064,Z 444.497,A -85,B 0,C 180,E1 -23367.794,E2 -23367.794} C_VEL
LIN {X 0,Y 209.651,Z 431.259,A -85,B 0,C 180,E1 -23368.35,E2 -23368.35} C_VEL
LIN {X 0,Y 211.772,Z 402.03,A -85,B 0,C 180,E1 -23369.221,E2 -23369.221} C_VEL
LIN {X 0,Y 206.244,Z 390.213,A -85,B 0,C 180,E1 -23371.883,E2 -23371.883} C_VEL
LIN {X 0,Y 202.303,Z 382.889,A -85,B 0,C 180,E1 -23373.917,E2 -23373.917} C_VEL
LIN {X 0,Y 196.414,Z 374.128,A -85,B 0,C 180,E1 -23377.192,E2 -23377.192} C_VEL
LIN {X 0,Y 193.571,Z 370.179,A -85,B 0,C 180,E1 -23378.947,E2 -23378.947} C_VEL
LIN {X 0,Y 191.35,Z 367.009,A -85,B 0,C 180,E1 -23380.454,E2 -23380.454} C_VEL
LIN {X 0,Y 188.218,Z 362.757,A -85,B 0,C 180,E1 -23382.777,E2 -23382.777} C_VEL
LIN {X 0,Y 185.583,Z 359.475,A -85,B 0,C 180,E1 -23384.944,E2 -23384.944} C_VEL
LIN {X 0,Y 184.638,Z 358.02,A -85,B 0,C 180,E1 -23385.817,E2 -23385.817} C_VEL
LIN {X 0,Y 181.868,Z 355.127,A -85,B 0,C 180,E1 -23388.489,E2 -23388.489} C_VEL
LIN {X 0,Y 180.502,Z 352.642,A -85,B 0,C 180,E1 -23390.139,E2 -23390.139} C_VEL
LIN {X 0,Y 177.513,Z 349.91,A -85,B 0,C 180,E1 -23394.142,E2 -23394.142} C_VEL
LIN {X 0,Y 176.305,Z 347.16,A -85,B 0,C 180,E1 -23396.573,E2 -23396.573} C_VEL
LIN {X 0,Y 174.103,Z 345.96,A -85,B 0,C 180,E1 -23402.314,E2 -23402.314} C_VEL
LIN {X 0,Y 173.717,Z 345.878,A -85,B 0,C 180,E1 -23409.313,E2 -23409.313} C_VEL
LIN {X 0,Y 176.18,Z 347.346,A -85,B 0,C 180,E1 -23416.909,E2 -23416.909} C_VEL
LIN {X 0,Y 177.388,Z 350.246,A -85,B 0,C 180,E1 -23419.405,E2 -23419.405} C_VEL
LIN {X 0,Y 179.654,Z 352.36,A -85,B 0,C 180,E1 -23422.574,E2 -23422.574} C_VEL
LIN {X 0,Y 180.718,Z 353.22,A -85,B 0,C 180,E1 -23423.825,E2 -23423.825} C_VEL
LIN {X 0,Y 182.515,Z 356.169,A -85,B 0,C 180,E1 -23425.882,E2 -23425.882} C_VEL
LIN {X 0,Y 185.952,Z 360.652,A -85,B 0,C 180,E1 -23429.113,E2 -23429.113} C_VEL
LIN {X 0,Y 189.844,Z 366.604,A -85,B 0,C 180,E1 -23432.271,E2 -23432.271} C_VEL
LIN {X 0,Y 193.459,Z 372.46,A -85,B 0,C 180,E1 -23434.831,E2 -23434.831} C_VEL
LIN {X 0,Y 196.981,Z 378.427,A -85,B 0,C 180,E1 -23437.053,E2 -23437.053} C_VEL
LIN {X 0,Y 201.348,Z 386.408,A -85,B 0,C 180,E1 -23439.565,E2 -23439.565} C_VEL
LIN {X 0,Y 206.091,Z 395.96,A -85,B 0,C 180,E1 -23442.061,E2 -23442.061} C_VEL
LIN {X 0,Y 210.858,Z 407.371,A -85,B 0,C 180,E1 -23444.423,E2 -23444.423} C_VEL
LIN {X 0,Y 211.374,Z 409.239,A -85,B 0,C 180,E1 -23444.699,E2 -23444.699} C_VEL
LIN {X 0,Y 208.66,Z 444.754,A -85,B 0,C 180,E1 -23445.798,E2 -23445.798} C_VEL
LIN {X 0,Y 206.719,Z 457.784,A -85,B 0,C 180,E1 -23446.494,E2 -23446.494} C_VEL
LIN {X 0,Y 203.821,Z 470.216,A -85,B 0,C 180,E1 -23447.417,E2 -23447.417} C_VEL
LIN {X 0,Y 200.559,Z 481.294,A -85,B 0,C 180,E1 -23448.595,E2 -23448.595} C_VEL
LIN {X 0,Y 196.364,Z 492.822,A -85,B 0,C 180,E1 -23450.229,E2 -23450.229} C_VEL
LIN {X 0,Y 191.803,Z 503.226,A -85,B 0,C 180,E1 -23452.142,E2 -23452.142} C_VEL
LIN {X 0,Y 187.221,Z 512.608,A -85,B 0,C 180,E1 -23454.422,E2 -23454.422} C_VEL
LIN {X 0,Y 181.955,Z 521.684,A -85,B 0,C 180,E1 -23457.268,E2 -23457.268} C_VEL
LIN {X 0,Y 179.867,Z 525.012,A -85,B 0,C 180,E1 -23458.539,E2 -23458.539} C_VEL
LIN {X 0,Y 177.141,Z 528.348,A -85,B 0,C 180,E1 -23459.853,E2 -23459.853} C_VEL
LIN {X 0,Y 171.274,Z 533.328,A -85,B 0,C 180,E1 -23461.92,E2 -23461.92} C_VEL
LIN {X 0,Y 165.588,Z 537.62,A -85,B 0,C 180,E1 -23464.261,E2 -23464.261} C_VEL
LIN {X 0,Y 163.213,Z 539.806,A -85,B 0,C 180,E1 -23465.981,E2 -23465.981} C_VEL
LIN {X 0,Y 160.264,Z 543.217,A -85,B 0,C 180,E1 -23469.465,E2 -23469.465} C_VEL
LIN {X 0,Y 158.546,Z 545.031,A -85,B 0,C 180,E1 -23471.926,E2 -23471.926} C_VEL
LIN {X 0,Y 156.232,Z 547.41,A -85,B 0,C 180,E1 -23477.004,E2 -23477.004} C_VEL
LIN {X 0,Y 154.979,Z 548.259,A -85,B 0,C 180,E1 -23482.183,E2 -23482.183} C_VEL
LIN {X 0,Y 154.747,Z 547.497,A -85,B 0,C 180,E1 -23487.399,E2 -23487.399} C_VEL
LIN {X 0,Y 154.867,Z 546.537,A -85,B 0,C 180,E1 -23490.002,E2 -23490.002} C_VEL
LIN {X 0,Y 154.743,Z 545.154,A -85,B 0,C 180,E1 -23492.605,E2 -23492.605} C_VEL
LIN {X 0,Y 154.898,Z 542.223,A -85,B 0,C 180,E1 -23496.515,E2 -23496.515} C_VEL
LIN {X 0,Y 155.391,Z 538.222,A -85,B 0,C 180,E1 -23500.425,E2 -23500.425} C_VEL
LIN {X 0,Y 156.567,Z 532.023,A -85,B 0,C 180,E1 -23504.96,E2 -23504.96} C_VEL
LIN {X 0,Y 158.386,Z 525.249,A -85,B 0,C 180,E1 -23508.768,E2 -23508.768} C_VEL
LIN {X 0,Y 160.372,Z 518.332,A -85,B 0,C 180,E1 -23511.872,E2 -23511.872} C_VEL
LIN {X 0,Y 162.189,Z 511.264,A -85,B 0,C 180,E1 -23514.497,E2 -23514.497} C_VEL
LIN {X 0,Y 164.764,Z 501.904,A -85,B 0,C 180,E1 -23517.295,E2 -23517.295} C_VEL
LIN {X 0,Y 167.514,Z 490.909,A -85,B 0,C 180,E1 -23519.884,E2 -23519.884} C_VEL
LIN {X 0,Y 170.086,Z 480.168,A -85,B 0,C 180,E1 -23521.794,E2 -23521.794} C_VEL
LIN {X 0,Y 172.301,Z 468.311,A -85,B 0,C 180,E1 -23523.414,E2 -23523.414} C_VEL
LIN {X 0,Y 174.067,Z 455.829,A -85,B 0,C 180,E1 -23524.654,E2 -23524.654} C_VEL
LIN {X 0,Y 175.308,Z 443.506,A -85,B 0,C 180,E1 -23525.455,E2 -23525.455} C_VEL
LIN {X 0,Y 177.686,Z 394.475,A -85,B 0,C 180,E1 -23527.346,E2 -23527.346} C_VEL
LIN {X 0,Y 176.083,Z 378.323,A -85,B 0,C 180,E1 -23528.436,E2 -23528.436} C_VEL
LIN {X 0,Y 170.779,Z 363.816,A -85,B 0,C 180,E1 -23530.304,E2 -23530.304} C_VEL
LIN {X 0,Y 165.246,Z 351.276,A -85,B 0,C 180,E1 -23532.282,E2 -23532.282} C_VEL
LIN {X 0,Y 160.863,Z 342.776,A -85,B 0,C 180,E1 -23533.901,E2 -23533.901} C_VEL
LIN {X 0,Y 159.221,Z 339.989,A -85,B 0,C 180,E1 -23534.517,E2 -23534.517} C_VEL
LIN {X 0,Y 157.607,Z 337.466,A -85,B 0,C 180,E1 -23535.128,E2 -23535.128} C_VEL
LIN {X 0,Y 157.223,Z 335.904,A -85,B 0,C 180,E1 -23535.397,E2 -23535.397} C_VEL
LIN {X 0,Y 157.211,Z 335.9,A -85,B 0,C 180,E1 -23541.254,E2 -23541.254} C_VEL
LIN {X 0,Y 157.284,Z 335.891,A -85,B 0,C 180,E1 -23544.486,E2 -23544.486} C_VEL
LIN {X 0,Y 157.289,Z 335.89,A -85,B 0,C 180,E1 -23548.103,E2 -23548.103} C_VEL
LIN {X 0,Y 157.315,Z 335.885,A -85,B 0,C 180,E1 -23553.464,E2 -23553.464} C_VEL
LIN {X 0,Y 157.367,Z 335.855,A -85,B 0,C 180,E1 -23559.701,E2 -23559.701} C_VEL
LIN {X 0,Y 157.425,Z 335.874,A -85,B 0,C 180,E1 -23564.462,E2 -23564.462} C_VEL
LIN {X 0,Y 157.693,Z 335.809,A -85,B 0,C 180,E1 -23569.73,E2 -23569.73} C_VEL
LIN {X 0,Y 157.768,Z 335.804,A -85,B 0,C 180,E1 -23572.319,E2 -23572.319} C_VEL
LIN {X 0,Y 158.252,Z 335.751,A -85,B 0,C 180,E1 -23579.999,E2 -23579.999} C_VEL
LIN {X 0,Y 157.766,Z 335.829,A -85,B 0,C 180,E1 -23587.679,E2 -23587.679} C_VEL
LIN {X 0,Y 157.638,Z 335.84,A -85,B 0,C 180,E1 -23591.227,E2 -23591.227} C_VEL
LIN {X 0,Y 157.423,Z 335.835,A -85,B 0,C 180,E1 -23595.537,E2 -23595.537} C_VEL
LIN {X 0,Y 157.318,Z 335.888,A -85,B 0,C 180,E1 -23600.939,E2 -23600.939} C_VEL
LIN {X 0,Y 157.314,Z 335.852,A -85,B 0,C 180,E1 -23606.679,E2 -23606.679} C_VEL
LIN {X 0,Y 157.272,Z 335.888,A -85,B 0,C 180,E1 -23612.428,E2 -23612.428} C_VEL
LIN {X 0,Y 157.264,Z 335.872,A -85,B 0,C 180,E1 -23616.444,E2 -23616.444} C_VEL
LIN {X 0,Y 157.195,Z 335.898,A -85,B 0,C 180,E1 -23622.115,E2 -23622.115} C_VEL
LIN {X 0,Y 157.195,Z 335.88,A -85,B 0,C 180,E1 -23627.881,E2 -23627.881} C_VEL
LIN {X 0,Y 157.27,Z 335.883,A -85,B 0,C 180,E1 -23633.549,E2 -23633.549} C_VEL
LIN {X 0,Y 157.348,Z 335.928,A -85,B 0,C 180,E1 -23639.17,E2 -23639.17} C_VEL
LIN {X 0,Y 158.265,Z 338.615,A -85,B 0,C 180,E1 -23639.595,E2 -23639.595} C_VEL
LIN {X 0,Y 159.993,Z 341.015,A -85,B 0,C 180,E1 -23640.223,E2 -23640.223} C_VEL
LIN {X 0,Y 167.898,Z 354.427,A -85,B 0,C 180,E1 -23643.003,E2 -23643.003} C_VEL
LIN {X 0,Y 175.14,Z 368.776,A -85,B 0,C 180,E1 -23645.368,E2 -23645.368} C_VEL
LIN {X 0,Y 178.434,Z 378.282,A -85,B 0,C 180,E1 -23646.504,E2 -23646.504} C_VEL
LIN {X 0,Y 175.857,Z 429.9,A -85,B 0,C 180,E1 -23648.43,E2 -23648.43} C_VEL
LIN {X 0,Y 174.737,Z 443.423,A -85,B 0,C 180,E1 -23649.162,E2 -23649.162} C_VEL
LIN {X 0,Y 173.255,Z 456.046,A -85,B 0,C 180,E1 -23650.292,E2 -23650.292} C_VEL
LIN {X 0,Y 171.244,Z 467.867,A -85,B 0,C 180,E1 -23651.762,E2 -23651.762} C_VEL
LIN {X 0,Y 168.864,Z 479.626,A -85,B 0,C 180,E1 -23653.756,E2 -23653.756} C_VEL
LIN {X 0,Y 166.196,Z 490.76,A -85,B 0,C 180,E1 -23656.205,E2 -23656.205} C_VEL
LIN {X 0,Y 163.663,Z 500.23,A -85,B 0,C 180,E1 -23658.856,E2 -23658.856} C_VEL
LIN {X 0,Y 161.193,Z 508.747,A -85,B 0,C 180,E1 -23661.852,E2 -23661.852} C_VEL
LIN {X 0,Y 158.799,Z 517.046,A -85,B 0,C 180,E1 -23665.556,E2 -23665.556} C_VEL
LIN {X 0,Y 157.031,Z 523.724,A -85,B 0,C 180,E1 -23669.357,E2 -23669.357} C_VEL
LIN {X 0,Y 155.674,Z 529.814,A -85,B 0,C 180,E1 -23673.881,E2 -23673.881} C_VEL
LIN {X 0,Y 154.883,Z 533.787,A -85,B 0,C 180,E1 -23677.821,E2 -23677.821} C_VEL
LIN {X 0,Y 154.505,Z 535.842,A -85,B 0,C 180,E1 -23680.481,E2 -23680.481} C_VEL
LIN {X 0,Y 154.382,Z 537.474,A -85,B 0,C 180,E1 -23683.154,E2 -23683.154} C_VEL
LIN {X 0,Y 154.638,Z 539.149,A -85,B 0,C 180,E1 -23687.37,E2 -23687.37} C_VEL
LIN {X 0,Y 155.22,Z 539.767,A -85,B 0,C 180,E1 -23691.234,E2 -23691.234} C_VEL
LIN {X 0,Y 155.947,Z 539.714,A -85,B 0,C 180,E1 -23693.926,E2 -23693.926} C_VEL
LIN {X 0,Y 156.959,Z 539.2,A -85,B 0,C 180,E1 -23696.597,E2 -23696.597} C_VEL
LIN {X 0,Y 158.208,Z 538.261,A -85,B 0,C 180,E1 -23699.249,E2 -23699.249} C_VEL
LIN {X 0,Y 159.777,Z 536.906,A -85,B 0,C 180,E1 -23701.856,E2 -23701.856} C_VEL
LIN {X 0,Y 162.676,Z 533.983,A -85,B 0,C 180,E1 -23705.675,E2 -23705.675} C_VEL
LIN {X 0,Y 166.234,Z 529.947,A -85,B 0,C 180,E1 -23709.355,E2 -23709.355} C_VEL
LIN {X 0,Y 170.402,Z 524.658,A -85,B 0,C 180,E1 -23712.881,E2 -23712.881} C_VEL
LIN {X 0,Y 175.148,Z 517.909,A -85,B 0,C 180,E1 -23716.239,E2 -23716.239} C_VEL
LIN {X 0,Y 180.546,Z 509.464,A -85,B 0,C 180,E1 -23719.378,E2 -23719.378} C_VEL
LIN {X 0,Y 185.379,Z 500.735,A -85,B 0,C 180,E1 -23721.871,E2 -23721.871} C_VEL
LIN {X 0,Y 189.999,Z 491.216,A -85,B 0,C 180,E1 -23723.952,E2 -23723.952} C_VEL
LIN {X 0,Y 194.316,Z 480.401,A -85,B 0,C 180,E1 -23725.822,E2 -23725.822} C_VEL
LIN {X 0,Y 198.281,Z 468.682,A -85,B 0,C 180,E1 -23727.327,E2 -23727.327} C_VEL
LIN {X 0,Y 201.278,Z 457.115,A -85,B 0,C 180,E1 -23728.446,E2 -23728.446} C_VEL
LIN {X 0,Y 203.716,Z 443.783,A -85,B 0,C 180,E1 -23729.364,E2 -23729.364} C_VEL
LIN {X 0,Y 205.277,Z 430.719,A -85,B 0,C 180,E1 -23729.898,E2 -23729.898} C_VEL
LIN {X 0,Y 207.24,Z 404.77,A -85,B 0,C 180,E1 -23730.665,E2 -23730.665} C_VEL
LIN {X 0,Y 202.285,Z 394.036,A -85,B 0,C 180,E1 -23733.224,E2 -23733.224} C_VEL
LIN {X 0,Y 199.038,Z 388.055,A -85,B 0,C 180,E1 -23735.001,E2 -23735.001} C_VEL
LIN {X 0,Y 193.716,Z 379.874,A -85,B 0,C 180,E1 -23738.139,E2 -23738.139} C_VEL
LIN {X 0,Y 189.246,Z 373.332,A -85,B 0,C 180,E1 -23741.194,E2 -23741.194} C_VEL
LIN {X 0,Y 186.226,Z 369.158,A -85,B 0,C 180,E1 -23743.541,E2 -23743.541} C_VEL
LIN {X 0,Y 183.462,Z 365.391,A -85,B 0,C 180,E1 -23745.971,E2 -23745.971} C_VEL
LIN {X 0,Y 182.418,Z 364.215,A -85,B 0,C 180,E1 -23746.954,E2 -23746.954} C_VEL
LIN {X 0,Y 179.885,Z 361.024,A -85,B 0,C 180,E1 -23749.65,E2 -23749.65} C_VEL
LIN {X 0,Y 179.076,Z 359.458,A -85,B 0,C 180,E1 -23750.704,E2 -23750.704} C_VEL
LIN {X 0,Y 176.267,Z 356.703,A -85,B 0,C 180,E1 -23754.674,E2 -23754.674} C_VEL
LIN {X 0,Y 174.979,Z 353.995,A -85,B 0,C 180,E1 -23757.4,E2 -23757.4} C_VEL
LIN {X 0,Y 173.22,Z 353.008,A -85,B 0,C 180,E1 -23762.326,E2 -23762.326} C_VEL
LIN {X 0,Y 172.844,Z 352.937,A -85,B 0,C 180,E1 -23769.361,E2 -23769.361} C_VEL
LIN {X 0,Y 175.025,Z 354.39,A -85,B 0,C 180,E1 -23776.443,E2 -23776.443} C_VEL
LIN {X 0,Y 176.41,Z 357.425,A -85,B 0,C 180,E1 -23779.331,E2 -23779.331} C_VEL
LIN {X 0,Y 179.223,Z 359.963,A -85,B 0,C 180,E1 -23783.19,E2 -23783.19} C_VEL
LIN {X 0,Y 184.111,Z 367.107,A -85,B 0,C 180,E1 -23788.382,E2 -23788.382} C_VEL
LIN {X 0,Y 187.714,Z 372.839,A -85,B 0,C 180,E1 -23791.464,E2 -23791.464} C_VEL
LIN {X 0,Y 191.193,Z 378.755,A -85,B 0,C 180,E1 -23794.072,E2 -23794.072} C_VEL
LIN {X 0,Y 195.51,Z 386.344,A -85,B 0,C 180,E1 -23796.897,E2 -23796.897} C_VEL
LIN {X 0,Y 201.119,Z 397.488,A -85,B 0,C 180,E1 -23800.172,E2 -23800.172} C_VEL
LIN {X 0,Y 205.75,Z 408.471,A -85,B 0,C 180,E1 -23802.663,E2 -23802.663} C_VEL
LIN {X 0,Y 206.787,Z 411.161,A -85,B 0,C 180,E1 -23803.2,E2 -23803.2} C_VEL
LIN {X 0,Y 204.177,Z 444.742,A -85,B 0,C 180,E1 -23804.274,E2 -23804.274} C_VEL
LIN {X 0,Y 202.136,Z 457.848,A -85,B 0,C 180,E1 -23804.977,E2 -23804.977} C_VEL
LIN {X 0,Y 198.989,Z 470.759,A -85,B 0,C 180,E1 -23805.949,E2 -23805.949} C_VEL
LIN {X 0,Y 195.342,Z 482.435,A -85,B 0,C 180,E1 -23807.231,E2 -23807.231} C_VEL
LIN {X 0,Y 191.009,Z 493.711,A -85,B 0,C 180,E1 -23808.879,E2 -23808.879} C_VEL
LIN {X 0,Y 186.288,Z 503.917,A -85,B 0,C 180,E1 -23810.811,E2 -23810.811} C_VEL
LIN {X 0,Y 181.529,Z 513.09,A -85,B 0,C 180,E1 -23813.126,E2 -23813.126} C_VEL
LIN {X 0,Y 176.899,Z 520.692,A -85,B 0,C 180,E1 -23815.522,E2 -23815.522} C_VEL
LIN {X 0,Y 171.881,Z 528.16,A -85,B 0,C 180,E1 -23818.581,E2 -23818.581} C_VEL
LIN {X 0,Y 167.014,Z 535.083,A -85,B 0,C 180,E1 -23822.429,E2 -23822.429} C_VEL
LIN {X 0,Y 163.213,Z 539.806,A -85,B 0,C 180,E1 -23825.981,E2 -23825.981} C_VEL
LIN {X 0,Y 160.937,Z 541.805,A -85,B 0,C 180,E1 -23827.787,E2 -23827.787} C_VEL
LIN {X 0,Y 155.768,Z 544.463,A -85,B 0,C 180,E1 -23830.698,E2 -23830.698} C_VEL
LIN {X 0,Y 151.003,Z 546.383,A -85,B 0,C 180,E1 -23833.859,E2 -23833.859} C_VEL
LIN {X 0,Y 149.422,Z 547.152,A -85,B 0,C 180,E1 -23835.998,E2 -23835.998} C_VEL
LIN {X 0,Y 148.481,Z 547.877,A -85,B 0,C 180,E1 -23839.089,E2 -23839.089} C_VEL
LIN {X 0,Y 147.692,Z 547.821,A -85,B 0,C 180,E1 -23844.541,E2 -23844.541} C_VEL
LIN {X 0,Y 147.678,Z 547.003,A -85,B 0,C 180,E1 -23848.024,E2 -23848.024} C_VEL
LIN {X 0,Y 147.767,Z 546.223,A -85,B 0,C 180,E1 -23850.002,E2 -23850.002} C_VEL
LIN {X 0,Y 147.647,Z 544.778,A -85,B 0,C 180,E1 -23852.731,E2 -23852.731} C_VEL
LIN {X 0,Y 147.816,Z 541.786,A -85,B 0,C 180,E1 -23856.829,E2 -23856.829} C_VEL
LIN {X 0,Y 148.367,Z 537.708,A -85,B 0,C 180,E1 -23860.925,E2 -23860.925} C_VEL
LIN {X 0,Y 149.663,Z 531.406,A -85,B 0,C 180,E1 -23865.667,E2 -23865.667} C_VEL
LIN {X 0,Y 151.644,Z 524.541,A -85,B 0,C 180,E1 -23869.636,E2 -23869.636} C_VEL
LIN {X 0,Y 153.787,Z 517.522,A -85,B 0,C 180,E1 -23872.86,E2 -23872.86} C_VEL
LIN {X 0,Y 155.622,Z 510.63,A -85,B 0,C 180,E1 -23875.483,E2 -23875.483} C_VEL
LIN {X 0,Y 158.392,Z 500.812,A -85,B 0,C 180,E1 -23878.491,E2 -23878.491} C_VEL
LIN {X 0,Y 161.383,Z 489.546,A -85,B 0,C 180,E1 -23881.143,E2 -23881.143} C_VEL
LIN {X 0,Y 164.045,Z 478.507,A -85,B 0,C 180,E1 -23883.111,E2 -23883.111} C_VEL
LIN {X 0,Y 166.401,Z 466.255,A -85,B 0,C 180,E1 -23884.765,E2 -23884.765} C_VEL
LIN {X 0,Y 168.155,Z 453.901,A -85,B 0,C 180,E1 -23885.952,E2 -23885.952} C_VEL
LIN {X 0,Y 169.377,Z 440.715,A -85,B 0,C 180,E1 -23886.754,E2 -23886.754} C_VEL
LIN {X 0,Y 171.639,Z 395.29,A -85,B 0,C 180,E1 -23888.542,E2 -23888.542} C_VEL
LIN {X 0,Y 170.223,Z 380.553,A -85,B 0,C 180,E1 -23889.585,E2 -23889.585} C_VEL
LIN {X 0,Y 165.19,Z 366.601,A -85,B 0,C 180,E1 -23891.481,E2 -23891.481} C_VEL
LIN {X 0,Y 160.038,Z 354.819,A -85,B 0,C 180,E1 -23893.45,E2 -23893.45} C_VEL
LIN {X 0,Y 155.768,Z 346.497,A -85,B 0,C 180,E1 -23895.14,E2 -23895.14} C_VEL
LIN {X 0,Y 152.337,Z 341.092,A -85,B 0,C 180,E1 -23896.519,E2 -23896.519} C_VEL
LIN {X 0,Y 150.596,Z 338.522,A -85,B 0,C 180,E1 -23897.244,E2 -23897.244} C_VEL
LIN {X 0,Y 150.147,Z 336.787,A -85,B 0,C 180,E1 -23897.55,E2 -23897.55} C_VEL
LIN {X 0,Y 150.185,Z 336.777,A -85,B 0,C 180,E1 -23902.708,E2 -23902.708} C_VEL
LIN {X 0,Y 150.214,Z 336.773,A -85,B 0,C 180,E1 -23907.372,E2 -23907.372} C_VEL
LIN {X 0,Y 150.244,Z 336.765,A -85,B 0,C 180,E1 -23912.723,E2 -23912.723} C_VEL
LIN {X 0,Y 150.291,Z 336.737,A -85,B 0,C 180,E1 -23919.275,E2 -23919.275} C_VEL
LIN {X 0,Y 150.33,Z 336.755,A -85,B 0,C 180,E1 -23923.709,E2 -23923.709} C_VEL
LIN {X 0,Y 150.613,Z 336.693,A -85,B 0,C 180,E1 -23929.242,E2 -23929.242} C_VEL
LIN {X 0,Y 150.69,Z 336.682,A -85,B 0,C 180,E1 -23931.956,E2 -23931.956} C_VEL
LIN {X 0,Y 151.212,Z 336.627,A -85,B 0,C 180,E1 -23939.999,E2 -23939.999} C_VEL
LIN {X 0,Y 150.704,Z 336.71,A -85,B 0,C 180,E1 -23948.042,E2 -23948.042} C_VEL
LIN {X 0,Y 150.58,Z 336.717,A -85,B 0,C 180,E1 -23951.43,E2 -23951.43} C_VEL
LIN {X 0,Y 150.326,Z 336.72,A -85,B 0,C 180,E1 -23956.29,E2 -23956.29} C_VEL
LIN {X 0,Y 150.29,Z 336.762,A -85,B 0,C 180,E1 -23960.724,E2 -23960.724} C_VEL
LIN {X 0,Y 150.243,Z 336.729,A -85,B 0,C 180,E1 -23967.276,E2 -23967.276} C_VEL
LIN {X 0,Y 150.212,Z 336.768,A -85,B 0,C 180,E1 -23972.626,E2 -23972.626} C_VEL
LIN {X 0,Y 150.173,Z 336.745,A -85,B 0,C 180,E1 -23977.473,E2 -23977.473} C_VEL
LIN {X 0,Y 150.139,Z 336.772,A -85,B 0,C 180,E1 -23981.496,E2 -23981.496} C_VEL
LIN {X 0,Y 150.129,Z 336.77,A -85,B 0,C 180,E1 -23985.394,E2 -23985.394} C_VEL
LIN {X 0,Y 150.143,Z 336.763,A -85,B 0,C 180,E1 -23989.053,E2 -23989.053} C_VEL
LIN {X 0,Y 150.185,Z 336.774,A -85,B 0,C 180,E1 -23992.704,E2 -23992.704} C_VEL
LIN {X 0,Y 150.204,Z 336.767,A -85,B 0,C 180,E1 -23996.961,E2 -23996.961} C_VEL
LIN {X 0,Y 151.214,Z 339.608,A -85,B 0,C 180,E1 -23997.493,E2 -23997.493} C_VEL
LIN {X 0,Y 153.046,Z 341.894,A -85,B 0,C 180,E1 -23998.22,E2 -23998.22} C_VEL
LIN {X 0,Y 160.616,Z 354.49,A -85,B 0,C 180,E1 -24001.155,E2 -24001.155} C_VEL
LIN {X 0,Y 166.344,Z 365.156,A -85,B 0,C 180,E1 -24003.189,E2 -24003.189} C_VEL
LIN {X 0,Y 170.592,Z 374.518,A -85,B 0,C 180,E1 -24004.657,E2 -24004.657} C_VEL
LIN {X 0,Y 172.457,Z 380.703,A -85,B 0,C 180,E1 -24005.376,E2 -24005.376} C_VEL
LIN {X 0,Y 169.255,Z 436.605,A -85,B 0,C 180,E1 -24007.541,E2 -24007.541} C_VEL
LIN {X 0,Y 167.823,Z 449.906,A -85,B 0,C 180,E1 -24008.502,E2 -24008.502} C_VEL
LIN {X 0,Y 165.954,Z 462.417,A -85,B 0,C 180,E1 -24009.872,E2 -24009.872} C_VEL
LIN {X 0,Y 163.866,Z 473.559,A -85,B 0,C 180,E1 -24011.558,E2 -24011.558} C_VEL
LIN {X 0,Y 161.141,Z 485.294,A -85,B 0,C 180,E1 -24013.888,E2 -24013.888} C_VEL
LIN {X 0,Y 158.339,Z 495.627,A -85,B 0,C 180,E1 -24016.522,E2 -24016.522} C_VEL
LIN {X 0,Y 155.63,Z 505.02,A -85,B 0,C 180,E1 -24019.591,E2 -24019.591} C_VEL
LIN {X 0,Y 152.867,Z 514.101,A -85,B 0,C 180,E1 -24023.398,E2 -24023.398} C_VEL
LIN {X 0,Y 150.708,Z 521.419,A -85,B 0,C 180,E1 -24027.325,E2 -24027.325} C_VEL
LIN {X 0,Y 149.17,Z 527.266,A -85,B 0,C 180,E1 -24031.347,E2 -24031.347} C_VEL
LIN {X 0,Y 148.216,Z 531.865,A -85,B 0,C 180,E1 -24035.439,E2 -24035.439} C_VEL
LIN {X 0,Y 147.507,Z 535.386,A -85,B 0,C 180,E1 -24039.597,E2 -24039.597} C_VEL
LIN {X 0,Y 147.286,Z 537.886,A -85,B 0,C 180,E1 -24043.8,E2 -24043.8} C_VEL
LIN {X 0,Y 147.564,Z 539.325,A -85,B 0,C 180,E1 -24047.725,E2 -24047.725} C_VEL
LIN {X 0,Y 148.333,Z 539.997,A -85,B 0,C 180,E1 -24052.271,E2 -24052.271} C_VEL
LIN {X 0,Y 150.003,Z 539.504,A -85,B 0,C 180,E1 -24057.104,E2 -24057.104} C_VEL
LIN {X 0,Y 151.747,Z 538.297,A -85,B 0,C 180,E1 -24060.624,E2 -24060.624} C_VEL
LIN {X 0,Y 155.011,Z 535.507,A -85,B 0,C 180,E1 -24065.305,E2 -24065.305} C_VEL
LIN {X 0,Y 159.167,Z 531.194,A -85,B 0,C 180,E1 -24069.807,E2 -24069.807} C_VEL
LIN {X 0,Y 163.47,Z 526.219,A -85,B 0,C 180,E1 -24073.459,E2 -24073.459} C_VEL
LIN {X 0,Y 168.311,Z 519.872,A -85,B 0,C 180,E1 -24076.944,E2 -24076.944} C_VEL
LIN {X 0,Y 172.558,Z 513.821,A -85,B 0,C 180,E1 -24079.471,E2 -24079.471} C_VEL
LIN {X 0,Y 177.783,Z 505.415,A -85,B 0,C 180,E1 -24082.24,E2 -24082.24} C_VEL
LIN {X 0,Y 183.174,Z 495.379,A -85,B 0,C 180,E1 -24084.735,E2 -24084.735} C_VEL
LIN {X 0,Y 188.011,Z 484.72,A -85,B 0,C 180,E1 -24086.757,E2 -24086.757} C_VEL
LIN {X 0,Y 192.04,Z 474.09,A -85,B 0,C 180,E1 -24088.302,E2 -24088.302} C_VEL
LIN {X 0,Y 195.572,Z 462.396,A -85,B 0,C 180,E1 -24089.589,E2 -24089.589} C_VEL
LIN {X 0,Y 198.523,Z 448.938,A -85,B 0,C 180,E1 -24090.667,E2 -24090.667} C_VEL
LIN {X 0,Y 200.485,Z 435.8,A -85,B 0,C 180,E1 -24091.334,E2 -24091.334} C_VEL
LIN {X 0,Y 202.796,Z 407.565,A -85,B 0,C 180,E1 -24092.188,E2 -24092.188} C_VEL
LIN {X 0,Y 198.838,Z 398.726,A -85,B 0,C 180,E1 -24094.387,E2 -24094.387} C_VEL
LIN {X 0,Y 195.755,Z 393.01,A -85,B 0,C 180,E1 -24096.178,E2 -24096.178} C_VEL
LIN {X 0,Y 190.855,Z 385.245,A -85,B 0,C 180,E1 -24099.269,E2 -24099.269} C_VEL
LIN {X 0,Y 186.933,Z 379.358,A -85,B 0,C 180,E1 -24102.13,E2 -24102.13} C_VEL
LIN {X 0,Y 184.059,Z 375.313,A -85,B 0,C 180,E1 -24104.498,E2 -24104.498} C_VEL
LIN {X 0,Y 181.221,Z 371.206,A -85,B 0,C 180,E1 -24107.187,E2 -24107.187} C_VEL
LIN {X 0,Y 178.506,Z 367.915,A -85,B 0,C 180,E1 -24110.142,E2 -24110.142} C_VEL
LIN {X 0,Y 177.567,Z 366.173,A -85,B 0,C 180,E1 -24111.408,E2 -24111.408} C_VEL
LIN {X 0,Y 174.948,Z 363.304,A -85,B 0,C 180,E1 -24115.392,E2 -24115.392} C_VEL
LIN {X 0,Y 173.95,Z 360.979,A -85,B 0,C 180,E1 -24117.685,E2 -24117.685} C_VEL
LIN {X 0,Y 172.338,Z 360.047,A -85,B 0,C 180,E1 -24122.338,E2 -24122.338} C_VEL
LIN {X 0,Y 171.971,Z 359.997,A -85,B 0,C 180,E1 -24129.409,E2 -24129.409} C_VEL
LIN {X 0,Y 173.873,Z 361.285,A -85,B 0,C 180,E1 -24135.904,E2 -24135.904} C_VEL
LIN {X 0,Y 175.334,Z 364.425,A -85,B 0,C 180,E1 -24139.079,E2 -24139.079} C_VEL
LIN {X 0,Y 177.716,Z 366.599,A -85,B 0,C 180,E1 -24142.488,E2 -24142.488} C_VEL
LIN {X 0,Y 182.146,Z 373.326,A -85,B 0,C 180,E1 -24147.486,E2 -24147.486} C_VEL
LIN {X 0,Y 185.641,Z 379.154,A -85,B 0,C 180,E1 -24150.658,E2 -24150.658} C_VEL
LIN {X 0,Y 188.709,Z 384.547,A -85,B 0,C 180,E1 -24153.095,E2 -24153.095} C_VEL
LIN {X 0,Y 192.94,Z 392.443,A -85,B 0,C 180,E1 -24156.055,E2 -24156.055} C_VEL
LIN {X 0,Y 197.912,Z 402.739,A -85,B 0,C 180,E1 -24159.132,E2 -24159.132} C_VEL
LIN {X 0,Y 202.087,Z 412.993,A -85,B 0,C 180,E1 -24161.525,E2 -24161.525} C_VEL
LIN {X 0,Y 202.384,Z 413.895,A -85,B 0,C 180,E1 -24161.696,E2 -24161.696} C_VEL
LIN {X 0,Y 199.859,Z 444.606,A -85,B 0,C 180,E1 -24162.677,E2 -24162.677} C_VEL
LIN {X 0,Y 197.674,Z 458.015,A -85,B 0,C 180,E1 -24163.395,E2 -24163.395} C_VEL
LIN {X 0,Y 194.606,Z 470.271,A -85,B 0,C 180,E1 -24164.318,E2 -24164.318} C_VEL
LIN {X 0,Y 190.801,Z 482.017,A -85,B 0,C 180,E1 -24165.588,E2 -24165.588} C_VEL
LIN {X 0,Y 186.313,Z 493.331,A -85,B 0,C 180,E1 -24167.239,E2 -24167.239} C_VEL
LIN {X 0,Y 181.413,Z 503.571,A -85,B 0,C 180,E1 -24169.179,E2 -24169.179} C_VEL
LIN {X 0,Y 176.915,Z 511.947,A -85,B 0,C 180,E1 -24171.271,E2 -24171.271} C_VEL
LIN {X 0,Y 171.108,Z 521.073,A -85,B 0,C 180,E1 -24174.179,E2 -24174.179} C_VEL
LIN {X 0,Y 165.872,Z 528.436,A -85,B 0,C 180,E1 -24177.305,E2 -24177.305} C_VEL
LIN {X 0,Y 160.752,Z 535.245,A -85,B 0,C 180,E1 -24181.258,E2 -24181.258} C_VEL
LIN {X 0,Y 156.53,Z 540.105,A -85,B 0,C 180,E1 -24185.139,E2 -24185.139} C_VEL
LIN {X 0,Y 153.623,Z 543.231,A -85,B 0,C 180,E1 -24188.534,E2 -24188.534} C_VEL
LIN {X 0,Y 151.795,Z 544.98,A -85,B 0,C 180,E1 -24191.092,E2 -24191.092} C_VEL
LIN {X 0,Y 149.422,Z 547.152,A -85,B 0,C 180,E1 -24195.998,E2 -24195.998} C_VEL
LIN {X 0,Y 148.061,Z 547.754,A -85,B 0,C 180,E1 -24198.198,E2 -24198.198} C_VEL
LIN {X 0,Y 144.462,Z 547.969,A -85,B 0,C 180,E1 -24201.813,E2 -24201.813} C_VEL
LIN {X 0,Y 141.755,Z 547.535,A -85,B 0,C 180,E1 -24204.819,E2 -24204.819} C_VEL
LIN {X 0,Y 140.661,Z 546.928,A -85,B 0,C 180,E1 -24207.18,E2 -24207.18} C_VEL
LIN {X 0,Y 140.587,Z 546.653,A -85,B 0,C 180,E1 -24207.982,E2 -24207.982} C_VEL
LIN {X 0,Y 140.597,Z 545.261,A -85,B 0,C 180,E1 -24211.291,E2 -24211.291} C_VEL
LIN {X 0,Y 140.761,Z 541.333,A -85,B 0,C 180,E1 -24217.173,E2 -24217.173} C_VEL
LIN {X 0,Y 141.368,Z 537.177,A -85,B 0,C 180,E1 -24221.473,E2 -24221.473} C_VEL
LIN {X 0,Y 142.801,Z 530.791,A -85,B 0,C 180,E1 -24226.441,E2 -24226.441} C_VEL
LIN {X 0,Y 144.933,Z 523.833,A -85,B 0,C 180,E1 -24230.585,E2 -24230.585} C_VEL
LIN {X 0,Y 147.616,Z 515.073,A -85,B 0,C 180,E1 -24234.622,E2 -24234.622} C_VEL
LIN {X 0,Y 150.33,Z 506.066,A -85,B 0,C 180,E1 -24237.875,E2 -24237.875} C_VEL
LIN {X 0,Y 153.188,Z 496.157,A -85,B 0,C 180,E1 -24240.693,E2 -24240.693} C_VEL
LIN {X 0,Y 155.343,Z 488.176,A -85,B 0,C 180,E1 -24242.499,E2 -24242.499} C_VEL
LIN {X 0,Y 158.065,Z 476.837,A -85,B 0,C 180,E1 -24244.537,E2 -24244.537} C_VEL
LIN {X 0,Y 160.352,Z 465.311,A -85,B 0,C 180,E1 -24246.085,E2 -24246.085} C_VEL
LIN {X 0,Y 162.145,Z 452.983,A -85,B 0,C 180,E1 -24247.264,E2 -24247.264} C_VEL
LIN {X 0,Y 163.436,Z 439.292,A -85,B 0,C 180,E1 -24248.085,E2 -24248.085} C_VEL
LIN {X 0,Y 165.666,Z 396.018,A -85,B 0,C 180,E1 -24249.831,E2 -24249.831} C_VEL
LIN {X 0,Y 164.504,Z 382.884,A -85,B 0,C 180,E1 -24250.788,E2 -24250.788} C_VEL
LIN {X 0,Y 159.486,Z 368.95,A -85,B 0,C 180,E1 -24252.807,E2 -24252.807} C_VEL
LIN {X 0,Y 154.097,Z 356.66,A -85,B 0,C 180,E1 -24255.032,E2 -24255.032} C_VEL
LIN {X 0,Y 150.48,Z 349.8,A -85,B 0,C 180,E1 -24256.573,E2 -24256.573} C_VEL
LIN {X 0,Y 147.829,Z 345.838,A -85,B 0,C 180,E1 -24257.705,E2 -24257.705} C_VEL
LIN {X 0,Y 145.379,Z 342.034,A -85,B 0,C 180,E1 -24258.816,E2 -24258.816} C_VEL
LIN {X 0,Y 143.555,Z 339.487,A -85,B 0,C 180,E1 -24259.661,E2 -24259.661} C_VEL
LIN {X 0,Y 143.07,Z 337.668,A -85,B 0,C 180,E1 -24259.987,E2 -24259.987} C_VEL
LIN {X 0,Y 143.165,Z 337.652,A -85,B 0,C 180,E1 -24266.571,E2 -24266.571} C_VEL
LIN {X 0,Y 143.189,Z 337.646,A -85,B 0,C 180,E1 -24272.069,E2 -24272.069} C_VEL
LIN {X 0,Y 143.232,Z 337.617,A -85,B 0,C 180,E1 -24278.798,E2 -24278.798} C_VEL
LIN {X 0,Y 143.267,Z 337.629,A -85,B 0,C 180,E1 -24282.882,E2 -24282.882} C_VEL
LIN {X 0,Y 143.539,Z 337.578,A -85,B 0,C 180,E1 -24288.705,E2 -24288.705} C_VEL
LIN {X 0,Y 143.615,Z 337.559,A -85,B 0,C 180,E1 -24291.557,E2 -24291.557} C_VEL
LIN {X 0,Y 144.169,Z 337.502,A -85,B 0,C 180,E1 -24299.999,E2 -24299.999} C_VEL
LIN {X 0,Y 143.626,Z 337.593,A -85,B 0,C 180,E1 -24308.441,E2 -24308.441} C_VEL
LIN {X 0,Y 143.505,Z 337.594,A -85,B 0,C 180,E1 -24311.618,E2 -24311.618} C_VEL
LIN {X 0,Y 143.264,Z 337.605,A -85,B 0,C 180,E1 -24317.117,E2 -24317.117} C_VEL
LIN {X 0,Y 143.231,Z 337.643,A -85,B 0,C 180,E1 -24321.201,E2 -24321.201} C_VEL
LIN {X 0,Y 143.187,Z 337.606,A -85,B 0,C 180,E1 -24327.929,E2 -24327.929} C_VEL
LIN {X 0,Y 143.142,Z 337.65,A -85,B 0,C 180,E1 -24333.415,E2 -24333.415} C_VEL
LIN {X 0,Y 143.057,Z 337.632,A -85,B 0,C 180,E1 -24339.691,E2 -24339.691} C_VEL
LIN {X 0,Y 143.055,Z 337.663,A -85,B 0,C 180,E1 -24343.455,E2 -24343.455} C_VEL
LIN {X 0,Y 143.042,Z 337.64,A -85,B 0,C 180,E1 -24347.475,E2 -24347.475} C_VEL
LIN {X 0,Y 143.082,Z 337.663,A -85,B 0,C 180,E1 -24351.803,E2 -24351.803} C_VEL
LIN {X 0,Y 143.128,Z 337.814,A -85,B 0,C 180,E1 -24354.528,E2 -24354.528} C_VEL
LIN {X 0,Y 144.103,Z 340.468,A -85,B 0,C 180,E1 -24355.076,E2 -24355.076} C_VEL
LIN {X 0,Y 146.125,Z 342.913,A -85,B 0,C 180,E1 -24355.976,E2 -24355.976} C_VEL
LIN {X 0,Y 148.475,Z 346.455,A -85,B 0,C 180,E1 -24357.02,E2 -24357.02} C_VEL
LIN {X 0,Y 156.781,Z 360.303,A -85,B 0,C 180,E1 -24360.427,E2 -24360.427} C_VEL
LIN {X 0,Y 163.949,Z 374.773,A -85,B 0,C 180,E1 -24363.115,E2 -24363.115} C_VEL
LIN {X 0,Y 166.483,Z 381.919,A -85,B 0,C 180,E1 -24364.095,E2 -24364.095} C_VEL
LIN {X 0,Y 163.232,Z 436.543,A -85,B 0,C 180,E1 -24366.259,E2 -24366.259} C_VEL
LIN {X 0,Y 161.737,Z 449.801,A -85,B 0,C 180,E1 -24367.229,E2 -24367.229} C_VEL
LIN {X 0,Y 159.888,Z 461.83,A -85,B 0,C 180,E1 -24368.567,E2 -24368.567} C_VEL
LIN {X 0,Y 157.51,Z 473.997,A -85,B 0,C 180,E1 -24370.447,E2 -24370.447} C_VEL
LIN {X 0,Y 154.625,Z 485.856,A -85,B 0,C 180,E1 -24372.892,E2 -24372.892} C_VEL
LIN {X 0,Y 151.73,Z 495.993,A -85,B 0,C 180,E1 -24375.581,E2 -24375.581} C_VEL
LIN {X 0,Y 149.177,Z 504.502,A -85,B 0,C 180,E1 -24378.448,E2 -24378.448} C_VEL
LIN {X 0,Y 146.206,Z 513.724,A -85,B 0,C 180,E1 -24382.401,E2 -24382.401} C_VEL
LIN {X 0,Y 143.883,Z 521.143,A -85,B 0,C 180,E1 -24386.497,E2 -24386.497} C_VEL
LIN {X 0,Y 142.465,Z 526.171,A -85,B 0,C 180,E1 -24389.997,E2 -24389.997} C_VEL
LIN {X 0,Y 141.381,Z 530.81,A -85,B 0,C 180,E1 -24394.036,E2 -24394.036} C_VEL
LIN {X 0,Y 140.529,Z 534.822,A -85,B 0,C 180,E1 -24398.626,E2 -24398.626} C_VEL
LIN {X 0,Y 140.23,Z 536.778,A -85,B 0,C 180,E1 -24401.562,E2 -24401.562} C_VEL
LIN {X 0,Y 140.217,Z 538.262,A -85,B 0,C 180,E1 -24404.511,E2 -24404.511} C_VEL
LIN {X 0,Y 140.508,Z 539.504,A -85,B 0,C 180,E1 -24408.132,E2 -24408.132} C_VEL
LIN {X 0,Y 141.494,Z 540.215,A -85,B 0,C 180,E1 -24413.41,E2 -24413.41} C_VEL
LIN {X 0,Y 143.182,Z 539.734,A -85,B 0,C 180,E1 -24417.931,E2 -24417.931} C_VEL
LIN {X 0,Y 145.391,Z 538.339,A -85,B 0,C 180,E1 -24422.119,E2 -24422.119} C_VEL
LIN {X 0,Y 148.541,Z 535.803,A -85,B 0,C 180,E1 -24426.455,E2 -24426.455} C_VEL
LIN {X 0,Y 152.11,Z 532.425,A -85,B 0,C 180,E1 -24430.301,E2 -24430.301} C_VEL
LIN {X 0,Y 156.542,Z 527.767,A -85,B 0,C 180,E1 -24434.085,E2 -24434.085} C_VEL
LIN {X 0,Y 161.538,Z 521.733,A -85,B 0,C 180,E1 -24437.695,E2 -24437.695} C_VEL
LIN {X 0,Y 166.626,Z 514.92,A -85,B 0,C 180,E1 -24440.753,E2 -24440.753} C_VEL
LIN {X 0,Y 172.282,Z 506.354,A -85,B 0,C 180,E1 -24443.671,E2 -24443.671} C_VEL
LIN {X 0,Y 177.75,Z 496.833,A -85,B 0,C 180,E1 -24446.127,E2 -24446.127} C_VEL
LIN {X 0,Y 182.883,Z 486.096,A -85,B 0,C 180,E1 -24448.233,E2 -24448.233} C_VEL
LIN {X 0,Y 187.05,Z 475.731,A -85,B 0,C 180,E1 -24449.784,E2 -24449.784} C_VEL
LIN {X 0,Y 190.726,Z 464.529,A -85,B 0,C 180,E1 -24451.059,E2 -24451.059} C_VEL
LIN {X 0,Y 193.806,Z 451.883,A -85,B 0,C 180,E1 -24452.135,E2 -24452.135} C_VEL
LIN {X 0,Y 195.898,Z 439.442,A -85,B 0,C 180,E1 -24452.845,E2 -24452.845} C_VEL
LIN {X 0,Y 197.861,Z 419.354,A -85,B 0,C 180,E1 -24453.474,E2 -24453.474} C_VEL
LIN {X 0,Y 198.483,Z 410.395,A -85,B 0,C 180,E1 -24453.784,E2 -24453.784} C_VEL
LIN {X 0,Y 194.544,Z 401.519,A -85,B 0,C 180,E1 -24456.162,E2 -24456.162} C_VEL
LIN {X 0,Y 189.888,Z 393.467,A -85,B 0,C 180,E1 -24459.158,E2 -24459.158} C_VEL
LIN {X 0,Y 184.95,Z 385.734,A -85,B 0,C 180,E1 -24462.864,E2 -24462.864} C_VEL
LIN {X 0,Y 182.143,Z 381.675,A -85,B 0,C 180,E1 -24465.297,E2 -24465.297} C_VEL
LIN {X 0,Y 179.37,Z 377.62,A -85,B 0,C 180,E1 -24468.076,E2 -24468.076} C_VEL
LIN {X 0,Y 176.799,Z 374.146,A -85,B 0,C 180,E1 -24471.106,E2 -24471.106} C_VEL
LIN {X 0,Y 176.062,Z 372.856,A -85,B 0,C 180,E1 -24472.157,E2 -24472.157} C_VEL
LIN {X 0,Y 173.538,Z 369.713,A -85,B 0,C 180,E1 -24476.389,E2 -24476.389} C_VEL
LIN {X 0,Y 172.779,Z 367.884,A -85,B 0,C 180,E1 -24478.311,E2 -24478.311} C_VEL
LIN {X 0,Y 171.455,Z 367.094,A -85,B 0,C 180,E1 -24482.35,E2 -24482.35} C_VEL
LIN {X 0,Y 171.098,Z 367.058,A -85,B 0,C 180,E1 -24489.457,E2 -24489.457} C_VEL
LIN {X 0,Y 172.774,Z 368.267,A -85,B 0,C 180,E1 -24495.448,E2 -24495.448} C_VEL
LIN {X 0,Y 174.152,Z 371.284,A -85,B 0,C 180,E1 -24498.62,E2 -24498.62} C_VEL
LIN {X 0,Y 176.414,Z 373.594,A -85,B 0,C 180,E1 -24502.042,E2 -24502.042} C_VEL
LIN {X 0,Y 180.461,Z 379.994,A -85,B 0,C 180,E1 -24506.822,E2 -24506.822} C_VEL
LIN {X 0,Y 183.612,Z 385.458,A -85,B 0,C 180,E1 -24509.842,E2 -24509.842} C_VEL
LIN {X 0,Y 186.505,Z 390.814,A -85,B 0,C 180,E1 -24512.276,E2 -24512.276} C_VEL
LIN {X 0,Y 190.228,Z 398.112,A -85,B 0,C 180,E1 -24515.058,E2 -24515.058} C_VEL
LIN {X 0,Y 194.951,Z 408.329,A -85,B 0,C 180,E1 -24518.165,E2 -24518.165} C_VEL
LIN {X 0,Y 198.093,Z 416.409,A -85,B 0,C 180,E1 -24520.099,E2 -24520.099} C_VEL
LIN {X 0,Y 195.72,Z 444.294,A -85,B 0,C 180,E1 -24521,E2 -24521} C_VEL
LIN {X 0,Y 193.426,Z 457.939,A -85,B 0,C 180,E1 -24521.728,E2 -24521.728} C_VEL
LIN {X 0,Y 190.063,Z 470.785,A -85,B 0,C 180,E1 -24522.703,E2 -24522.703} C_VEL
LIN {X 0,Y 185.834,Z 483.166,A -85,B 0,C 180,E1 -24524.068,E2 -24524.068} C_VEL
LIN {X 0,Y 181.207,Z 494.234,A -85,B 0,C 180,E1 -24525.727,E2 -24525.727} C_VEL
LIN {X 0,Y 175.565,Z 505.206,A -85,B 0,C 180,E1 -24527.896,E2 -24527.896} C_VEL
LIN {X 0,Y 170.417,Z 514.086,A -85,B 0,C 180,E1 -24530.269,E2 -24530.269} C_VEL
LIN {X 0,Y 164.48,Z 522.802,A -85,B 0,C 180,E1 -24533.262,E2 -24533.262} C_VEL
LIN {X 0,Y 159.095,Z 529.788,A -85,B 0,C 180,E1 -24536.486,E2 -24536.486} C_VEL
LIN {X 0,Y 154.548,Z 535.393,A -85,B 0,C 180,E1 -24539.988,E2 -24539.988} C_VEL
LIN {X 0,Y 150.437,Z 539.837,A -85,B 0,C 180,E1 -24543.656,E2 -24543.656} C_VEL
LIN {X 0,Y 147.031,Z 543.233,A -85,B 0,C 180,E1 -24547.521,E2 -24547.521} C_VEL
LIN {X 0,Y 143.534,Z 546.246,A -85,B 0,C 180,E1 -24552.918,E2 -24552.918} C_VEL
LIN {X 0,Y 141.487,Z 547.709,A -85,B 0,C 180,E1 -24558.542,E2 -24558.542} C_VEL
LIN {X 0,Y 140.623,Z 547.573,A -85,B 0,C 180,E1 -24564.266,E2 -24564.266} C_VEL
LIN {X 0,Y 140.587,Z 546.653,A -85,B 0,C 180,E1 -24567.982,E2 -24567.982} C_VEL
LIN {X 0,Y 139.937,Z 545.707,A -85,B 0,C 180,E1 -24570.34,E2 -24570.34} C_VEL
LIN {X 0,Y 138.361,Z 544.447,A -85,B 0,C 180,E1 -24572.643,E2 -24572.643} C_VEL
LIN {X 0,Y 134.808,Z 541.135,A -85,B 0,C 180,E1 -24577.266,E2 -24577.266} C_VEL
LIN {X 0,Y 134.025,Z 539.063,A -85,B 0,C 180,E1 -24579.647,E2 -24579.647} C_VEL
LIN {X 0,Y 134.068,Z 538.303,A -85,B 0,C 180,E1 -24580.442,E2 -24580.442} C_VEL
LIN {X 0,Y 135.171,Z 533.156,A -85,B 0,C 180,E1 -24585.071,E2 -24585.071} C_VEL
LIN {X 0,Y 137.062,Z 526.833,A -85,B 0,C 180,E1 -24589.471,E2 -24589.471} C_VEL
LIN {X 0,Y 139.64,Z 518.88,A -85,B 0,C 180,E1 -24593.746,E2 -24593.746} C_VEL
LIN {X 0,Y 141.956,Z 511.353,A -85,B 0,C 180,E1 -24596.98,E2 -24596.98} C_VEL
LIN {X 0,Y 145.004,Z 501.87,A -85,B 0,C 180,E1 -24600.191,E2 -24600.191} C_VEL
LIN {X 0,Y 148.113,Z 490.996,A -85,B 0,C 180,E1 -24603.074,E2 -24603.074} C_VEL
LIN {X 0,Y 151.038,Z 480.482,A -85,B 0,C 180,E1 -24605.16,E2 -24605.16} C_VEL
LIN {X 0,Y 153.541,Z 468.88,A -85,B 0,C 180,E1 -24606.928,E2 -24606.928} C_VEL
LIN {X 0,Y 155.688,Z 455.752,A -85,B 0,C 180,E1 -24608.369,E2 -24608.369} C_VEL
LIN {X 0,Y 157.148,Z 443.265,A -85,B 0,C 180,E1 -24609.256,E2 -24609.256} C_VEL
LIN {X 0,Y 159.814,Z 397.297,A -85,B 0,C 180,E1 -24611.162,E2 -24611.162} C_VEL
LIN {X 0,Y 158.737,Z 384.916,A -85,B 0,C 180,E1 -24612.117,E2 -24612.117} C_VEL
LIN {X 0,Y 153.742,Z 371.032,A -85,B 0,C 180,E1 -24614.285,E2 -24614.285} C_VEL
LIN {X 0,Y 148.756,Z 359.645,A -85,B 0,C 180,E1 -24616.512,E2 -24616.512} C_VEL
LIN {X 0,Y 145.76,Z 354.059,A -85,B 0,C 180,E1 -24617.882,E2 -24617.882} C_VEL
LIN {X 0,Y 141.156,Z 347.028,A -85,B 0,C 180,E1 -24620.054,E2 -24620.054} C_VEL
LIN {X 0,Y 138.619,Z 343.199,A -85,B 0,C 180,E1 -24621.342,E2 -24621.342} C_VEL
LIN {X 0,Y 136.652,Z 340.667,A -85,B 0,C 180,E1 -24622.357,E2 -24622.357} C_VEL
LIN {X 0,Y 136.027,Z 338.542,A -85,B 0,C 180,E1 -24622.853,E2 -24622.853} C_VEL
LIN {X 0,Y 136.089,Z 338.53,A -85,B 0,C 180,E1 -24625.723,E2 -24625.723} C_VEL
LIN {X 0,Y 136.129,Z 338.524,A -85,B 0,C 180,E1 -24632.312,E2 -24632.312} C_VEL
LIN {X 0,Y 136.198,Z 338.492,A -85,B 0,C 180,E1 -24638.825,E2 -24638.825} C_VEL
LIN {X 0,Y 136.237,Z 338.514,A -85,B 0,C 180,E1 -24645.052,E2 -24645.052} C_VEL
LIN {X 0,Y 136.431,Z 338.467,A -85,B 0,C 180,E1 -24648.178,E2 -24648.178} C_VEL
LIN {X 0,Y 136.544,Z 338.437,A -85,B 0,C 180,E1 -24651.117,E2 -24651.117} C_VEL
LIN {X 0,Y 137.125,Z 338.377,A -85,B 0,C 180,E1 -24659.999,E2 -24659.999} C_VEL
LIN {X 0,Y 136.552,Z 338.474,A -85,B 0,C 180,E1 -24668.881,E2 -24668.881} C_VEL
LIN {X 0,Y 136.42,Z 338.473,A -85,B 0,C 180,E1 -24671.891,E2 -24671.891} C_VEL
LIN {X 0,Y 136.175,Z 338.496,A -85,B 0,C 180,E1 -24678.038,E2 -24678.038} C_VEL
LIN {X 0,Y 136.158,Z 338.523,A -85,B 0,C 180,E1 -24681.699,E2 -24681.699} C_VEL
LIN {X 0,Y 136.096,Z 338.49,A -85,B 0,C 180,E1 -24688.608,E2 -24688.608} C_VEL
LIN {X 0,Y 136.044,Z 338.529,A -85,B 0,C 180,E1 -24694.628,E2 -24694.628} C_VEL
LIN {X 0,Y 136.029,Z 338.504,A -85,B 0,C 180,E1 -24699.193,E2 -24699.193} C_VEL
LIN {X 0,Y 135.997,Z 338.542,A -85,B 0,C 180,E1 -24703.653,E2 -24703.653} C_VEL
LIN {X 0,Y 135.986,Z 338.518,A -85,B 0,C 180,E1 -24707.786,E2 -24707.786} C_VEL
LIN {X 0,Y 136.065,Z 338.644,A -85,B 0,C 180,E1 -24711.694,E2 -24711.694} C_VEL
LIN {X 0,Y 137.03,Z 341.397,A -85,B 0,C 180,E1 -24712.321,E2 -24712.321} C_VEL
LIN {X 0,Y 139.273,Z 344.008,A -85,B 0,C 180,E1 -24713.448,E2 -24713.448} C_VEL
LIN {X 0,Y 141.357,Z 347.2,A -85,B 0,C 180,E1 -24714.501,E2 -24714.501} C_VEL
LIN {X 0,Y 146.45,Z 354.902,A -85,B 0,C 180,E1 -24716.878,E2 -24716.878} C_VEL
LIN {X 0,Y 153.929,Z 368.303,A -85,B 0,C 180,E1 -24720.074,E2 -24720.074} C_VEL
LIN {X 0,Y 159.431,Z 380.047,A -85,B 0,C 180,E1 -24722.26,E2 -24722.26} C_VEL
LIN {X 0,Y 160.554,Z 383.422,A -85,B 0,C 180,E1 -24722.734,E2 -24722.734} C_VEL
LIN {X 0,Y 157.231,Z 436.974,A -85,B 0,C 180,E1 -24724.918,E2 -24724.918} C_VEL
LIN {X 0,Y 155.61,Z 450.637,A -85,B 0,C 180,E1 -24725.959,E2 -24725.959} C_VEL
LIN {X 0,Y 153.497,Z 463.373,A -85,B 0,C 180,E1 -24727.45,E2 -24727.45} C_VEL
LIN {X 0,Y 150.863,Z 475.956,A -85,B 0,C 180,E1 -24729.548,E2 -24729.548} C_VEL
LIN {X 0,Y 148.162,Z 486.357,A -85,B 0,C 180,E1 -24731.807,E2 -24731.807} C_VEL
LIN {X 0,Y 145.165,Z 496.315,A -85,B 0,C 180,E1 -24734.555,E2 -24734.555} C_VEL
LIN {X 0,Y 142.189,Z 505.64,A -85,B 0,C 180,E1 -24737.871,E2 -24737.871} C_VEL
LIN {X 0,Y 139.143,Z 514.686,A -85,B 0,C 180,E1 -24742.013,E2 -24742.013} C_VEL
LIN {X 0,Y 136.764,Z 521.971,A -85,B 0,C 180,E1 -24746.314,E2 -24746.314} C_VEL
LIN {X 0,Y 135.301,Z 526.883,A -85,B 0,C 180,E1 -24749.997,E2 -24749.997} C_VEL
LIN {X 0,Y 134.054,Z 532.186,A -85,B 0,C 180,E1 -24755.068,E2 -24755.068} C_VEL
LIN {X 0,Y 133.345,Z 535.331,A -85,B 0,C 180,E1 -24759.095,E2 -24759.095} C_VEL
LIN {X 0,Y 133.096,Z 537.217,A -85,B 0,C 180,E1 -24762.191,E2 -24762.191} C_VEL
LIN {X 0,Y 133.151,Z 538.628,A -85,B 0,C 180,E1 -24765.299,E2 -24765.299} C_VEL
LIN {X 0,Y 133.456,Z 539.679,A -85,B 0,C 180,E1 -24768.577,E2 -24768.577} C_VEL
LIN {X 0,Y 133.916,Z 540.246,A -85,B 0,C 180,E1 -24771.55,E2 -24771.55} C_VEL
LIN {X 0,Y 134.717,Z 540.401,A -85,B 0,C 180,E1 -24774.664,E2 -24774.664} C_VEL
LIN {X 0,Y 136.385,Z 539.963,A -85,B 0,C 180,E1 -24778.835,E2 -24778.835} C_VEL
LIN {X 0,Y 139.124,Z 538.356,A -85,B 0,C 180,E1 -24783.754,E2 -24783.754} C_VEL
LIN {X 0,Y 142.186,Z 536.073,A -85,B 0,C 180,E1 -24787.736,E2 -24787.736} C_VEL
LIN {X 0,Y 146.499,Z 532.235,A -85,B 0,C 180,E1 -24792.189,E2 -24792.189} C_VEL
LIN {X 0,Y 151.468,Z 527.215,A -85,B 0,C 180,E1 -24796.21,E2 -24796.21} C_VEL
LIN {X 0,Y 156.6,Z 521.281,A -85,B 0,C 180,E1 -24799.72,E2 -24799.72} C_VEL
LIN {X 0,Y 162.791,Z 513.378,A -85,B 0,C 180,E1 -24803.138,E2 -24803.138} C_VEL
LIN {X 0,Y 168.008,Z 505.607,A -85,B 0,C 180,E1 -24805.703,E2 -24805.703} C_VEL
LIN {X 0,Y 173.732,Z 495.791,A -85,B 0,C 180,E1 -24808.154,E2 -24808.154} C_VEL
LIN {X 0,Y 179.096,Z 484.792,A -85,B 0,C 180,E1 -24810.248,E2 -24810.248} C_VEL
LIN {X 0,Y 183.461,Z 474.096,A -85,B 0,C 180,E1 -24811.768,E2 -24811.768} C_VEL
LIN {X 0,Y 187.001,Z 463.152,A -85,B 0,C 180,E1 -24812.964,E2 -24812.964} C_VEL
LIN {X 0,Y 190.18,Z 449.756,A -85,B 0,C 180,E1 -24814.039,E2 -24814.039} C_VEL
LIN {X 0,Y 192.24,Z 437.143,A -85,B 0,C 180,E1 -24814.689,E2 -24814.689} C_VEL
LIN {X 0,Y 194.373,Z 413.299,A -85,B 0,C 180,E1 -24815.426,E2 -24815.426} C_VEL
LIN {X 0,Y 190.758,Z 405.237,A -85,B 0,C 180,E1 -24817.782,E2 -24817.782} C_VEL
LIN {X 0,Y 185.986,Z 397.003,A -85,B 0,C 180,E1 -24821.177,E2 -24821.177} C_VEL
LIN {X 0,Y 182.554,Z 391.529,A -85,B 0,C 180,E1 -24823.991,E2 -24823.991} C_VEL
LIN {X 0,Y 180.365,Z 388.166,A -85,B 0,C 180,E1 -24826.016,E2 -24826.016} C_VEL
LIN {X 0,Y 177.638,Z 384.088,A -85,B 0,C 180,E1 -24828.9,E2 -24828.9} C_VEL
LIN {X 0,Y 175.131,Z 380.324,A -85,B 0,C 180,E1 -24832.115,E2 -24832.115} C_VEL
LIN {X 0,Y 174.396,Z 379.33,A -85,B 0,C 180,E1 -24833.22,E2 -24833.22} C_VEL
LIN {X 0,Y 172.274,Z 376.276,A -85,B 0,C 180,E1 -24837.186,E2 -24837.186} C_VEL
LIN {X 0,Y 171.63,Z 374.782,A -85,B 0,C 180,E1 -24838.945,E2 -24838.945} C_VEL
LIN {X 0,Y 170.571,Z 374.141,A -85,B 0,C 180,E1 -24842.362,E2 -24842.362} C_VEL
LIN {X 0,Y 170.226,Z 374.114,A -85,B 0,C 180,E1 -24849.506,E2 -24849.506} C_VEL
LIN {X 0,Y 171.721,Z 375.308,A -85,B 0,C 180,E1 -24855.083,E2 -24855.083} C_VEL
LIN {X 0,Y 173.175,Z 378.418,A -85,B 0,C 180,E1 -24858.512,E2 -24858.512} C_VEL
LIN {X 0,Y 175.066,Z 380.441,A -85,B 0,C 180,E1 -24861.492,E2 -24861.492} C_VEL
LIN {X 0,Y 178.684,Z 386.377,A -85,B 0,C 180,E1 -24866.013,E2 -24866.013} C_VEL
LIN {X 0,Y 181.541,Z 391.598,A -85,B 0,C 180,E1 -24868.931,E2 -24868.931} C_VEL
LIN {X 0,Y 185.153,Z 398.584,A -85,B 0,C 180,E1 -24872.101,E2 -24872.101} C_VEL
LIN {X 0,Y 188.936,Z 406.757,A -85,B 0,C 180,E1 -24875.026,E2 -24875.026} C_VEL
LIN {X 0,Y 192.699,Z 415.666,A -85,B 0,C 180,E1 -24877.609,E2 -24877.609} C_VEL
LIN {X 0,Y 193.948,Z 419.074,A -85,B 0,C 180,E1 -24878.436,E2 -24878.436} C_VEL
LIN {X 0,Y 191.73,Z 444.266,A -85,B 0,C 180,E1 -24879.271,E2 -24879.271} C_VEL
LIN {X 0,Y 189.411,Z 457.549,A -85,B 0,C 180,E1 -24879.968,E2 -24879.968} C_VEL
LIN {X 0,Y 186.019,Z 470.3,A -85,B 0,C 180,E1 -24880.924,E2 -24880.924} C_VEL
LIN {X 0,Y 182.218,Z 481.182,A -85,B 0,C 180,E1 -24882.062,E2 -24882.062} C_VEL
LIN {X 0,Y 177.392,Z 492.577,A -85,B 0,C 180,E1 -24883.698,E2 -24883.698} C_VEL
LIN {X 0,Y 172.13,Z 502.875,A -85,B 0,C 180,E1 -24885.64,E2 -24885.64} C_VEL
LIN {X 0,Y 167.165,Z 511.307,A -85,B 0,C 180,E1 -24887.729,E2 -24887.729} C_VEL
LIN {X 0,Y 161.881,Z 519.115,A -85,B 0,C 180,E1 -24890.184,E2 -24890.184} C_VEL
LIN {X 0,Y 155.979,Z 526.769,A -85,B 0,C 180,E1 -24893.347,E2 -24893.347} C_VEL
LIN {X 0,Y 151.552,Z 532.024,A -85,B 0,C 180,E1 -24896.19,E2 -24896.19} C_VEL
LIN {X 0,Y 146.959,Z 537.142,A -85,B 0,C 180,E1 -24899.861,E2 -24899.861} C_VEL
LIN {X 0,Y 142.801,Z 541.144,A -85,B 0,C 180,E1 -24903.712,E2 -24903.712} C_VEL
LIN {X 0,Y 140.492,Z 543.225,A -85,B 0,C 180,E1 -24906.413,E2 -24906.413} C_VEL
LIN {X 0,Y 136.729,Z 546.168,A -85,B 0,C 180,E1 -24912.04,E2 -24912.04} C_VEL
LIN {X 0,Y 135.462,Z 547.058,A -85,B 0,C 180,E1 -24914.968,E2 -24914.968} C_VEL
LIN {X 0,Y 133.879,Z 547.613,A -85,B 0,C 180,E1 -24920.942,E2 -24920.942} C_VEL
LIN {X 0,Y 133.512,Z 546.654,A -85,B 0,C 180,E1 -24926.985,E2 -24926.985} C_VEL
LIN {X 0,Y 133.543,Z 545.236,A -85,B 0,C 180,E1 -24930.681,E2 -24930.681} C_VEL
LIN {X 0,Y 133.569,Z 542.037,A -85,B 0,C 180,E1 -24936.043,E2 -24936.043} C_VEL
LIN {X 0,Y 134.068,Z 538.303,A -85,B 0,C 180,E1 -24940.442,E2 -24940.442} C_VEL
LIN {X 0,Y 133.908,Z 535.957,A -85,B 0,C 180,E1 -24942.757,E2 -24942.757} C_VEL
LIN {X 0,Y 132.26,Z 531.588,A -85,B 0,C 180,E1 -24946.518,E2 -24946.518} C_VEL
LIN {X 0,Y 130.962,Z 526.536,A -85,B 0,C 180,E1 -24950.205,E2 -24950.205} C_VEL
LIN {X 0,Y 131.349,Z 523.117,A -85,B 0,C 180,E1 -24952.315,E2 -24952.315} C_VEL
LIN {X 0,Y 134.021,Z 515.364,A -85,B 0,C 180,E1 -24956.249,E2 -24956.249} C_VEL
LIN {X 0,Y 136.506,Z 507.938,A -85,B 0,C 180,E1 -24959.283,E2 -24959.283} C_VEL
LIN {X 0,Y 139.985,Z 497.306,A -85,B 0,C 180,E1 -24962.667,E2 -24962.667} C_VEL
LIN {X 0,Y 142.218,Z 489.629,A -85,B 0,C 180,E1 -24964.634,E2 -24964.634} C_VEL
LIN {X 0,Y 145.241,Z 478.754,A -85,B 0,C 180,E1 -24966.787,E2 -24966.787} C_VEL
LIN {X 0,Y 147.901,Z 466.728,A -85,B 0,C 180,E1 -24968.588,E2 -24968.588} C_VEL
LIN {X 0,Y 149.93,Z 454.461,A -85,B 0,C 180,E1 -24969.914,E2 -24969.914} C_VEL
LIN {X 0,Y 151.423,Z 441.098,A -85,B 0,C 180,E1 -24970.82,E2 -24970.82} C_VEL
LIN {X 0,Y 153.972,Z 397.47,A -85,B 0,C 180,E1 -24972.68,E2 -24972.68} C_VEL
LIN {X 0,Y 153.225,Z 387.594,A -85,B 0,C 180,E1 -24973.461,E2 -24973.461} C_VEL
LIN {X 0,Y 148.566,Z 374.253,A -85,B 0,C 180,E1 -24975.659,E2 -24975.659} C_VEL
LIN {X 0,Y 143.289,Z 361.999,A -85,B 0,C 180,E1 -24978.227,E2 -24978.227} C_VEL
LIN {X 0,Y 139.185,Z 355.248,A -85,B 0,C 180,E1 -24980.244,E2 -24980.244} C_VEL
LIN {X 0,Y 134.66,Z 348.384,A -85,B 0,C 180,E1 -24982.647,E2 -24982.647} C_VEL
LIN {X 0,Y 132.55,Z 345.263,A -85,B 0,C 180,E1 -24983.852,E2 -24983.852} C_VEL
LIN {X 0,Y 131.83,Z 344.25,A -85,B 0,C 180,E1 -24984.274,E2 -24984.274} C_VEL
LIN {X 0,Y 129.97,Z 342.127,A -85,B 0,C 180,E1 -24985.362,E2 -24985.362} C_VEL
LIN {X 0,Y 129.014,Z 339.413,A -85,B 0,C 180,E1 -24986.156,E2 -24986.156} C_VEL
LIN {X 0,Y 129.023,Z 339.413,A -85,B 0,C 180,E1 -24990.643,E2 -24990.643} C_VEL
LIN {X 0,Y 129.019,Z 339.411,A -85,B 0,C 180,E1 -24994.164,E2 -24994.164} C_VEL
LIN {X 0,Y 129.078,Z 339.387,A -85,B 0,C 180,E1 -24997.767,E2 -24997.767} C_VEL
LIN {X 0,Y 129.158,Z 339.395,A -85,B 0,C 180,E1 -25004.212,E2 -25004.212} C_VEL
LIN {X 0,Y 129.35,Z 339.35,A -85,B 0,C 180,E1 -25007.97,E2 -25007.97} C_VEL
LIN {X 0,Y 129.469,Z 339.317,A -85,B 0,C 180,E1 -25010.627,E2 -25010.627} C_VEL
LIN {X 0,Y 130.079,Z 339.252,A -85,B 0,C 180,E1 -25019.999,E2 -25019.999} C_VEL
LIN {X 0,Y 129.475,Z 339.355,A -85,B 0,C 180,E1 -25029.371,E2 -25029.371} C_VEL
LIN {X 0,Y 129.303,Z 339.349,A -85,B 0,C 180,E1 -25032.556,E2 -25032.556} C_VEL
LIN {X 0,Y 129.093,Z 339.391,A -85,B 0,C 180,E1 -25039.065,E2 -25039.065} C_VEL
LIN {X 0,Y 129.078,Z 339.404,A -85,B 0,C 180,E1 -25042.403,E2 -25042.403} C_VEL
LIN {X 0,Y 129.021,Z 339.375,A -85,B 0,C 180,E1 -25049.356,E2 -25049.356} C_VEL
LIN {X 0,Y 128.96,Z 339.406,A -85,B 0,C 180,E1 -25055.164,E2 -25055.164} C_VEL
LIN {X 0,Y 128.932,Z 339.399,A -85,B 0,C 180,E1 -25060.851,E2 -25060.851} C_VEL
LIN {X 0,Y 128.931,Z 339.396,A -85,B 0,C 180,E1 -25067.381,E2 -25067.381} C_VEL
LIN {X 0,Y 128.93,Z 339.398,A -85,B 0,C 180,E1 -25068.312,E2 -25068.312} C_VEL
LIN {X 0,Y 129.855,Z 342.141,A -85,B 0,C 180,E1 -25069.048,E2 -25069.048} C_VEL
LIN {X 0,Y 131.727,Z 344.21,A -85,B 0,C 180,E1 -25070.138,E2 -25070.138} C_VEL
LIN {X 0,Y 132.511,Z 345.191,A -85,B 0,C 180,E1 -25070.587,E2 -25070.587} C_VEL
LIN {X 0,Y 134.711,Z 348.475,A -85,B 0,C 180,E1 -25071.843,E2 -25071.843} C_VEL
LIN {X 0,Y 140.482,Z 356.958,A -85,B 0,C 180,E1 -25074.848,E2 -25074.848} C_VEL
LIN {X 0,Y 148.183,Z 370.474,A -85,B 0,C 180,E1 -25078.447,E2 -25078.447} C_VEL
LIN {X 0,Y 154.226,Z 383.505,A -85,B 0,C 180,E1 -25081.048,E2 -25081.048} C_VEL
LIN {X 0,Y 154.723,Z 385.579,A -85,B 0,C 180,E1 -25081.307,E2 -25081.307} C_VEL
LIN {X 0,Y 151.374,Z 436.862,A -85,B 0,C 180,E1 -25083.437,E2 -25083.437} C_VEL
LIN {X 0,Y 149.706,Z 450.323,A -85,B 0,C 180,E1 -25084.468,E2 -25084.468} C_VEL
LIN {X 0,Y 147.598,Z 462.754,A -85,B 0,C 180,E1 -25085.936,E2 -25085.936} C_VEL
LIN {X 0,Y 144.997,Z 474.759,A -85,B 0,C 180,E1 -25087.933,E2 -25087.933} C_VEL
LIN {X 0,Y 142.06,Z 485.794,A -85,B 0,C 180,E1 -25090.357,E2 -25090.357} C_VEL
LIN {X 0,Y 138.652,Z 496.635,A -85,B 0,C 180,E1 -25093.431,E2 -25093.431} C_VEL
LIN {X 0,Y 135.834,Z 505.1,A -85,B 0,C 180,E1 -25096.534,E2 -25096.534} C_VEL
LIN {X 0,Y 132.543,Z 514.282,A -85,B 0,C 180,E1 -25100.844,E2 -25100.844} C_VEL
LIN {X 0,Y 129.983,Z 521.672,A -85,B 0,C 180,E1 -25105.345,E2 -25105.345} C_VEL
LIN {X 0,Y 128.142,Z 527.594,A -85,B 0,C 180,E1 -25109.997,E2 -25109.997} C_VEL
LIN {X 0,Y 126.975,Z 532.416,A -85,B 0,C 180,E1 -25114.945,E2 -25114.945} C_VEL
LIN {X 0,Y 126.191,Z 535.835,A -85,B 0,C 180,E1 -25119.615,E2 -25119.615} C_VEL
LIN {X 0,Y 125.976,Z 537.629,A -85,B 0,C 180,E1 -25122.891,E2 -25122.891} C_VEL
LIN {X 0,Y 126.398,Z 539.848,A -85,B 0,C 180,E1 -25129.052,E2 -25129.052} C_VEL
LIN {X 0,Y 127.057,Z 540.492,A -85,B 0,C 180,E1 -25132.777,E2 -25132.777} C_VEL
LIN {X 0,Y 128.035,Z 540.583,A -85,B 0,C 180,E1 -25136.045,E2 -25136.045} C_VEL
LIN {X 0,Y 129.64,Z 540.186,A -85,B 0,C 180,E1 -25139.845,E2 -25139.845} C_VEL
LIN {X 0,Y 132.981,Z 538.35,A -85,B 0,C 180,E1 -25145.541,E2 -25145.541} C_VEL
LIN {X 0,Y 135.875,Z 536.354,A -85,B 0,C 180,E1 -25149.118,E2 -25149.118} C_VEL
LIN {X 0,Y 139.509,Z 533.384,A -85,B 0,C 180,E1 -25152.846,E2 -25152.846} C_VEL
LIN {X 0,Y 144.886,Z 528.45,A -85,B 0,C 180,E1 -25157.228,E2 -25157.228} C_VEL
LIN {X 0,Y 150.892,Z 521.986,A -85,B 0,C 180,E1 -25161.27,E2 -25161.27} C_VEL
LIN {X 0,Y 157.093,Z 514.519,A -85,B 0,C 180,E1 -25164.616,E2 -25164.616} C_VEL
LIN {X 0,Y 162.795,Z 506.55,A -85,B 0,C 180,E1 -25167.329,E2 -25167.329} C_VEL
LIN {X 0,Y 168.285,Z 497.751,A -85,B 0,C 180,E1 -25169.62,E2 -25169.62} C_VEL
LIN {X 0,Y 173.665,Z 487.515,A -85,B 0,C 180,E1 -25171.661,E2 -25171.661} C_VEL
LIN {X 0,Y 178.131,Z 477.38,A -85,B 0,C 180,E1 -25173.203,E2 -25173.203} C_VEL
LIN {X 0,Y 182.182,Z 466.109,A -85,B 0,C 180,E1 -25174.502,E2 -25174.502} C_VEL
LIN {X 0,Y 185.705,Z 452.944,A -85,B 0,C 180,E1 -25175.645,E2 -25175.645} C_VEL
LIN {X 0,Y 188.081,Z 439.991,A -85,B 0,C 180,E1 -25176.371,E2 -25176.371} C_VEL
LIN {X 0,Y 189.995,Z 421.864,A -85,B 0,C 180,E1 -25176.941,E2 -25176.941} C_VEL
LIN {X 0,Y 190.444,Z 416.302,A -85,B 0,C 180,E1 -25177.122,E2 -25177.122} C_VEL
LIN {X 0,Y 187.788,Z 410.347,A -85,B 0,C 180,E1 -25178.995,E2 -25178.995} C_VEL
LIN {X 0,Y 183.416,Z 402.482,A -85,B 0,C 180,E1 -25182.348,E2 -25182.348} C_VEL
LIN {X 0,Y 180.205,Z 397.271,A -85,B 0,C 180,E1 -25185.171,E2 -25185.171} C_VEL
LIN {X 0,Y 178.171,Z 394.003,A -85,B 0,C 180,E1 -25187.208,E2 -25187.208} C_VEL
LIN {X 0,Y 175.958,Z 390.545,A -85,B 0,C 180,E1 -25189.727,E2 -25189.727} C_VEL
LIN {X 0,Y 173.294,Z 386.275,A -85,B 0,C 180,E1 -25193.506,E2 -25193.506} C_VEL
LIN {X 0,Y 171.166,Z 383.181,A -85,B 0,C 180,E1 -25197.647,E2 -25197.647} C_VEL
LIN {X 0,Y 170.641,Z 381.78,A -85,B 0,C 180,E1 -25199.205,E2 -25199.205} C_VEL
LIN {X 0,Y 169.687,Z 381.189,A -85,B 0,C 180,E1 -25202.374,E2 -25202.374} C_VEL
LIN {X 0,Y 169.352,Z 381.177,A -85,B 0,C 180,E1 -25209.556,E2 -25209.556} C_VEL
LIN {X 0,Y 170.613,Z 382.147,A -85,B 0,C 180,E1 -25214.504,E2 -25214.504} C_VEL
LIN {X 0,Y 172.091,Z 385.39,A -85,B 0,C 180,E1 -25218.198,E2 -25218.198} C_VEL
LIN {X 0,Y 173.71,Z 387.203,A -85,B 0,C 180,E1 -25220.879,E2 -25220.879} C_VEL
LIN {X 0,Y 176.93,Z 392.777,A -85,B 0,C 180,E1 -25225.178,E2 -25225.178} C_VEL
LIN {X 0,Y 179.717,Z 398.111,A -85,B 0,C 180,E1 -25228.197,E2 -25228.197} C_VEL
LIN {X 0,Y 183.098,Z 405.151,A -85,B 0,C 180,E1 -25231.35,E2 -25231.35} C_VEL
LIN {X 0,Y 186.465,Z 412.853,A -85,B 0,C 180,E1 -25234.117,E2 -25234.117} C_VEL
LIN {X 0,Y 189.798,Z 421.291,A -85,B 0,C 180,E1 -25236.58,E2 -25236.58} C_VEL
LIN {X 0,Y 190.01,Z 421.925,A -85,B 0,C 180,E1 -25236.734,E2 -25236.734} C_VEL
LIN {X 0,Y 187.905,Z 444.228,A -85,B 0,C 180,E1 -25237.46,E2 -25237.46} C_VEL
LIN {X 0,Y 185.467,Z 457.711,A -85,B 0,C 180,E1 -25238.168,E2 -25238.168} C_VEL
LIN {X 0,Y 181.988,Z 470.271,A -85,B 0,C 180,E1 -25239.1,E2 -25239.1} C_VEL
LIN {X 0,Y 177.597,Z 482.326,A -85,B 0,C 180,E1 -25240.383,E2 -25240.383} C_VEL
LIN {X 0,Y 172.598,Z 493.48,A -85,B 0,C 180,E1 -25242.006,E2 -25242.006} C_VEL
LIN {X 0,Y 167.166,Z 503.56,A -85,B 0,C 180,E1 -25243.952,E2 -25243.952} C_VEL
LIN {X 0,Y 160.893,Z 513.464,A -85,B 0,C 180,E1 -25246.533,E2 -25246.533} C_VEL
LIN {X 0,Y 154.417,Z 522.215,A -85,B 0,C 180,E1 -25249.57,E2 -25249.57} C_VEL
LIN {X 0,Y 148.422,Z 529.248,A -85,B 0,C 180,E1 -25252.866,E2 -25252.866} C_VEL
LIN {X 0,Y 142.395,Z 535.689,A -85,B 0,C 180,E1 -25257.121,E2 -25257.121} C_VEL
LIN {X 0,Y 137.851,Z 539.971,A -85,B 0,C 180,E1 -25261.034,E2 -25261.034} C_VEL
LIN {X 0,Y 134.014,Z 543.218,A -85,B 0,C 180,E1 -25265.198,E2 -25265.198} C_VEL
LIN {X 0,Y 129.963,Z 546.089,A -85,B 0,C 180,E1 -25271.07,E2 -25271.07} C_VEL
LIN {X 0,Y 128.598,Z 546.919,A -85,B 0,C 180,E1 -25274.145,E2 -25274.145} C_VEL
LIN {X 0,Y 126.868,Z 547.396,A -85,B 0,C 180,E1 -25280.437,E2 -25280.437} C_VEL
LIN {X 0,Y 126.439,Z 546.361,A -85,B 0,C 180,E1 -25286.817,E2 -25286.817} C_VEL
LIN {X 0,Y 126.506,Z 545.206,A -85,B 0,C 180,E1 -25290.003,E2 -25290.003} C_VEL
LIN {X 0,Y 126.403,Z 542.677,A -85,B 0,C 180,E1 -25294.787,E2 -25294.787} C_VEL
LIN {X 0,Y 126.852,Z 539.112,A -85,B 0,C 180,E1 -25299.57,E2 -25299.57} C_VEL
LIN {X 0,Y 127.807,Z 534.399,A -85,B 0,C 180,E1 -25304.33,E2 -25304.33} C_VEL
LIN {X 0,Y 129.937,Z 527.279,A -85,B 0,C 180,E1 -25309.761,E2 -25309.761} C_VEL
LIN {X 0,Y 131.349,Z 523.117,A -85,B 0,C 180,E1 -25312.315,E2 -25312.315} C_VEL
LIN {X 0,Y 131.833,Z 519.54,A -85,B 0,C 180,E1 -25314.351,E2 -25314.351} C_VEL
LIN {X 0,Y 131.229,Z 513.281,A -85,B 0,C 180,E1 -25317.715,E2 -25317.715} C_VEL
LIN {X 0,Y 130.989,Z 506.514,A -85,B 0,C 180,E1 -25320.875,E2 -25320.875} C_VEL
LIN {X 0,Y 131.984,Z 502.07,A -85,B 0,C 180,E1 -25322.507,E2 -25322.507} C_VEL
LIN {X 0,Y 135.043,Z 492.262,A -85,B 0,C 180,E1 -25325.381,E2 -25325.381} C_VEL
LIN {X 0,Y 138.209,Z 482.147,A -85,B 0,C 180,E1 -25327.607,E2 -25327.607} C_VEL
LIN {X 0,Y 141.162,Z 470.216,A -85,B 0,C 180,E1 -25329.638,E2 -25329.638} C_VEL
LIN {X 0,Y 143.505,Z 457.744,A -85,B 0,C 180,E1 -25331.157,E2 -25331.157} C_VEL
LIN {X 0,Y 145.372,Z 443.88,A -85,B 0,C 180,E1 -25332.248,E2 -25332.248} C_VEL
LIN {X 0,Y 148.304,Z 398.378,A -85,B 0,C 180,E1 -25334.254,E2 -25334.254} C_VEL
LIN {X 0,Y 147.554,Z 389.381,A -85,B 0,C 180,E1 -25335.037,E2 -25335.037} C_VEL
LIN {X 0,Y 143.031,Z 376.299,A -85,B 0,C 180,E1 -25337.366,E2 -25337.366} C_VEL
LIN {X 0,Y 137.949,Z 364.64,A -85,B 0,C 180,E1 -25340.061,E2 -25340.061} C_VEL
LIN {X 0,Y 132.281,Z 355.739,A -85,B 0,C 180,E1 -25343.152,E2 -25343.152} C_VEL
LIN {X 0,Y 130.498,Z 353.132,A -85,B 0,C 180,E1 -25344.196,E2 -25344.196} C_VEL
LIN {X 0,Y 128.269,Z 349.782,A -85,B 0,C 180,E1 -25345.579,E2 -25345.579} C_VEL
LIN {X 0,Y 126.233,Z 347.112,A -85,B 0,C 180,E1 -25346.885,E2 -25346.885} C_VEL
LIN {X 0,Y 125.281,Z 345.486,A -85,B 0,C 180,E1 -25347.558,E2 -25347.558} C_VEL
LIN {X 0,Y 123.04,Z 343.345,A -85,B 0,C 180,E1 -25349.063,E2 -25349.063} C_VEL
LIN {X 0,Y 122.041,Z 340.948,A -85,B 0,C 180,E1 -25349.91,E2 -25349.91} C_VEL
LIN {X 0,Y 121.95,Z 340.292,A -85,B 0,C 180,E1 -25350.144,E2 -25350.144} C_VEL
LIN {X 0,Y 122.013,Z 340.272,A -85,B 0,C 180,E1 -25357.169,E2 -25357.169} C_VEL
LIN {X 0,Y 122.07,Z 340.269,A -85,B 0,C 180,E1 -25363.269,E2 -25363.269} C_VEL
LIN {X 0,Y 122.293,Z 340.231,A -85,B 0,C 180,E1 -25367.691,E2 -25367.691} C_VEL
LIN {X 0,Y 122.397,Z 340.197,A -85,B 0,C 180,E1 -25370.08,E2 -25370.08} C_VEL
LIN {X 0,Y 122.586,Z 340.212,A -85,B 0,C 180,E1 -25376.713,E2 -25376.713} C_VEL
LIN {X 0,Y 123.032,Z 340.128,A -85,B 0,C 180,E1 -25379.999,E2 -25379.999} C_VEL
LIN {X 0,Y 122.398,Z 340.225,A -85,B 0,C 180,E1 -25386.91,E2 -25386.91} C_VEL
LIN {X 0,Y 122.293,Z 340.223,A -85,B 0,C 180,E1 -25392.309,E2 -25392.309} C_VEL
LIN {X 0,Y 122.069,Z 340.236,A -85,B 0,C 180,E1 -25396.73,E2 -25396.73} C_VEL
LIN {X 0,Y 122.009,Z 340.281,A -85,B 0,C 180,E1 -25402.827,E2 -25402.827} C_VEL
LIN {X 0,Y 121.93,Z 340.264,A -85,B 0,C 180,E1 -25410.159,E2 -25410.159} C_VEL
LIN {X 0,Y 121.884,Z 340.273,A -85,B 0,C 180,E1 -25416.167,E2 -25416.167} C_VEL
LIN {X 0,Y 121.872,Z 340.284,A -85,B 0,C 180,E1 -25421.434,E2 -25421.434} C_VEL
LIN {X 0,Y 121.858,Z 340.369,A -85,B 0,C 180,E1 -25424.388,E2 -25424.388} C_VEL
LIN {X 0,Y 122.788,Z 342.978,A -85,B 0,C 180,E1 -25425.22,E2 -25425.22} C_VEL
LIN {X 0,Y 124.79,Z 345.187,A -85,B 0,C 180,E1 -25426.608,E2 -25426.608} C_VEL
LIN {X 0,Y 125.61,Z 346.036,A -85,B 0,C 180,E1 -25427.146,E2 -25427.146} C_VEL
LIN {X 0,Y 127.524,Z 349.107,A -85,B 0,C 180,E1 -25428.449,E2 -25428.449} C_VEL
LIN {X 0,Y 129.025,Z 350.871,A -85,B 0,C 180,E1 -25429.367,E2 -25429.367} C_VEL
LIN {X 0,Y 134.946,Z 359.674,A -85,B 0,C 180,E1 -25432.795,E2 -25432.795} C_VEL
LIN {X 0,Y 139.707,Z 367.706,A -85,B 0,C 180,E1 -25435.302,E2 -25435.302} C_VEL
LIN {X 0,Y 144.789,Z 377.434,A -85,B 0,C 180,E1 -25437.774,E2 -25437.774} C_VEL
LIN {X 0,Y 149.01,Z 386.759,A -85,B 0,C 180,E1 -25439.714,E2 -25439.714} C_VEL
LIN {X 0,Y 145.603,Z 436.999,A -85,B 0,C 180,E1 -25441.854,E2 -25441.854} C_VEL
LIN {X 0,Y 143.811,Z 450.787,A -85,B 0,C 180,E1 -25442.938,E2 -25442.938} C_VEL
LIN {X 0,Y 141.584,Z 463.209,A -85,B 0,C 180,E1 -25444.451,E2 -25444.451} C_VEL
LIN {X 0,Y 138.858,Z 475.141,A -85,B 0,C 180,E1 -25446.508,E2 -25446.508} C_VEL
LIN {X 0,Y 135.731,Z 486.317,A -85,B 0,C 180,E1 -25449.059,E2 -25449.059} C_VEL
LIN {X 0,Y 132.197,Z 496.954,A -85,B 0,C 180,E1 -25452.198,E2 -25452.198} C_VEL
LIN {X 0,Y 128.902,Z 506.225,A -85,B 0,C 180,E1 -25455.795,E2 -25455.795} C_VEL
LIN {X 0,Y 125.511,Z 515.241,A -85,B 0,C 180,E1 -25460.326,E2 -25460.326} C_VEL
LIN {X 0,Y 122.873,Z 522.496,A -85,B 0,C 180,E1 -25465.075,E2 -25465.075} C_VEL
LIN {X 0,Y 120.988,Z 528.275,A -85,B 0,C 180,E1 -25469.997,E2 -25469.997} C_VEL
LIN {X 0,Y 119.885,Z 532.597,A -85,B 0,C 180,E1 -25474.743,E2 -25474.743} C_VEL
LIN {X 0,Y 119.031,Z 536.308,A -85,B 0,C 180,E1 -25480.199,E2 -25480.199} C_VEL
LIN {X 0,Y 118.87,Z 538.042,A -85,B 0,C 180,E1 -25483.676,E2 -25483.676} C_VEL
LIN {X 0,Y 119.374,Z 540.026,A -85,B 0,C 180,E1 -25489.615,E2 -25489.615} C_VEL
LIN {X 0,Y 120.258,Z 540.722,A -85,B 0,C 180,E1 -25494.144,E2 -25494.144} C_VEL
LIN {X 0,Y 121.414,Z 540.766,A -85,B 0,C 180,E1 -25497.582,E2 -25497.582} C_VEL
LIN {X 0,Y 122.935,Z 540.407,A -85,B 0,C 180,E1 -25500.961,E2 -25500.961} C_VEL
LIN {X 0,Y 124.769,Z 539.6,A -85,B 0,C 180,E1 -25504.279,E2 -25504.279} C_VEL
LIN {X 0,Y 127.006,Z 538.344,A -85,B 0,C 180,E1 -25507.491,E2 -25507.491} C_VEL
LIN {X 0,Y 130.886,Z 535.736,A -85,B 0,C 180,E1 -25511.948,E2 -25511.948} C_VEL
LIN {X 0,Y 135.845,Z 531.813,A -85,B 0,C 180,E1 -25516.406,E2 -25516.406} C_VEL
LIN {X 0,Y 141.321,Z 526.785,A -85,B 0,C 180,E1 -25520.423,E2 -25520.423} C_VEL
LIN {X 0,Y 147.421,Z 520.385,A -85,B 0,C 180,E1 -25524.134,E2 -25524.134} C_VEL
LIN {X 0,Y 154.178,Z 512.295,A -85,B 0,C 180,E1 -25527.485,E2 -25527.485} C_VEL
LIN {X 0,Y 160.125,Z 503.951,A -85,B 0,C 180,E1 -25530.088,E2 -25530.088} C_VEL
LIN {X 0,Y 166.427,Z 493.713,A -85,B 0,C 180,E1 -25532.468,E2 -25532.468} C_VEL
LIN {X 0,Y 171.596,Z 483.479,A -85,B 0,C 180,E1 -25534.29,E2 -25534.29} C_VEL
LIN {X 0,Y 176.275,Z 472.249,A -85,B 0,C 180,E1 -25535.779,E2 -25535.779} C_VEL
LIN {X 0,Y 180.436,Z 459.464,A -85,B 0,C 180,E1 -25537.036,E2 -25537.036} C_VEL
LIN {X 0,Y 183.272,Z 447.18,A -85,B 0,C 180,E1 -25537.913,E2 -25537.913} C_VEL
LIN {X 0,Y 185.375,Z 433.137,A -85,B 0,C 180,E1 -25538.509,E2 -25538.509} C_VEL
LIN {X 0,Y 186.668,Z 419.453,A -85,B 0,C 180,E1 -25538.898,E2 -25538.898} C_VEL
LIN {X 0,Y 184.71,Z 415.069,A -85,B 0,C 180,E1 -25540.409,E2 -25540.409} C_VEL
LIN {X 0,Y 180.755,Z 407.706,A -85,B 0,C 180,E1 -25543.7,E2 -25543.7} C_VEL
LIN {X 0,Y 176.97,Z 401.239,A -85,B 0,C 180,E1 -25547.421,E2 -25547.421} C_VEL
LIN {X 0,Y 174.512,Z 397.258,A -85,B 0,C 180,E1 -25550.322,E2 -25550.322} C_VEL
LIN {X 0,Y 171.898,Z 392.925,A -85,B 0,C 180,E1 -25554.281,E2 -25554.281} C_VEL
LIN {X 0,Y 170.013,Z 389.925,A -85,B 0,C 180,E1 -25558.284,E2 -25558.284} C_VEL
LIN {X 0,Y 169.656,Z 388.772,A -85,B 0,C 180,E1 -25559.467,E2 -25559.467} C_VEL
LIN {X 0,Y 168.803,Z 388.23,A -85,B 0,C 180,E1 -25562.387,E2 -25562.387} C_VEL
LIN {X 0,Y 168.322,Z 388.101,A -85,B 0,C 180,E1 -25568.057,E2 -25568.057} C_VEL
LIN {X 0,Y 169.601,Z 389.234,A -85,B 0,C 180,E1 -25574.205,E2 -25574.205} C_VEL
LIN {X 0,Y 171.034,Z 392.346,A -85,B 0,C 180,E1 -25577.914,E2 -25577.914} C_VEL
LIN {X 0,Y 172.416,Z 394.016,A -85,B 0,C 180,E1 -25580.321,E2 -25580.321} C_VEL
LIN {X 0,Y 175.181,Z 399.092,A -85,B 0,C 180,E1 -25584.282,E2 -25584.282} C_VEL
LIN {X 0,Y 177.747,Z 404.332,A -85,B 0,C 180,E1 -25587.27,E2 -25587.27} C_VEL
LIN {X 0,Y 180.637,Z 410.622,A -85,B 0,C 180,E1 -25590.165,E2 -25590.165} C_VEL
LIN {X 0,Y 184.158,Z 419.189,A -85,B 0,C 180,E1 -25593.272,E2 -25593.272} C_VEL
LIN {X 0,Y 186.226,Z 424.75,A -85,B 0,C 180,E1 -25594.943,E2 -25594.943} C_VEL
LIN {X 0,Y 184.291,Z 444.168,A -85,B 0,C 180,E1 -25595.582,E2 -25595.582} C_VEL
LIN {X 0,Y 181.753,Z 457.722,A -85,B 0,C 180,E1 -25596.286,E2 -25596.286} C_VEL
LIN {X 0,Y 178.23,Z 470.041,A -85,B 0,C 180,E1 -25597.183,E2 -25597.183} C_VEL
LIN {X 0,Y 173.762,Z 481.909,A -85,B 0,C 180,E1 -25598.408,E2 -25598.408} C_VEL
LIN {X 0,Y 168.614,Z 493.098,A -85,B 0,C 180,E1 -25600.018,E2 -25600.018} C_VEL
LIN {X 0,Y 162.97,Z 503.221,A -85,B 0,C 180,E1 -25601.939,E2 -25601.939} C_VEL
LIN {X 0,Y 157.001,Z 512.342,A -85,B 0,C 180,E1 -25604.26,E2 -25604.26} C_VEL
LIN {X 0,Y 150.189,Z 521.248,A -85,B 0,C 180,E1 -25607.276,E2 -25607.276} C_VEL
LIN {X 0,Y 143.843,Z 528.442,A -85,B 0,C 180,E1 -25610.571,E2 -25610.571} C_VEL
LIN {X 0,Y 138.011,Z 534.383,A -85,B 0,C 180,E1 -25614.337,E2 -25614.337} C_VEL
LIN {X 0,Y 133.243,Z 538.782,A -85,B 0,C 180,E1 -25618.17,E2 -25618.17} C_VEL
LIN {X 0,Y 128.848,Z 542.283,A -85,B 0,C 180,E1 -25622.382,E2 -25622.382} C_VEL
LIN {X 0,Y 125.244,Z 544.806,A -85,B 0,C 180,E1 -25626.875,E2 -25626.875} C_VEL
LIN {X 0,Y 123.241,Z 546,A -85,B 0,C 180,E1 -25629.995,E2 -25629.995} C_VEL
LIN {X 0,Y 120.625,Z 547.162,A -85,B 0,C 180,E1 -25636.526,E2 -25636.526} C_VEL
LIN {X 0,Y 119.42,Z 546.82,A -85,B 0,C 180,E1 -25643.244,E2 -25643.244} C_VEL
LIN {X 0,Y 119.353,Z 546.046,A -85,B 0,C 180,E1 -25646.627,E2 -25646.627} C_VEL
LIN {X 0,Y 119.419,Z 544.852,A -85,B 0,C 180,E1 -25650.003,E2 -25650.003} C_VEL
LIN {X 0,Y 119.327,Z 542.249,A -85,B 0,C 180,E1 -25655.071,E2 -25655.071} C_VEL
LIN {X 0,Y 119.823,Z 538.604,A -85,B 0,C 180,E1 -25660.138,E2 -25660.138} C_VEL
LIN {X 0,Y 120.883,Z 533.805,A -85,B 0,C 180,E1 -25665.169,E2 -25665.169} C_VEL
LIN {X 0,Y 122.817,Z 527.724,A -85,B 0,C 180,E1 -25670.084,E2 -25670.084} C_VEL
LIN {X 0,Y 125.534,Z 520.132,A -85,B 0,C 180,E1 -25674.83,E2 -25674.83} C_VEL
LIN {X 0,Y 127.42,Z 514.922,A -85,B 0,C 180,E1 -25677.468,E2 -25677.468} C_VEL
LIN {X 0,Y 130.322,Z 506.892,A -85,B 0,C 180,E1 -25680.821,E2 -25680.821} C_VEL
LIN {X 0,Y 131.984,Z 502.07,A -85,B 0,C 180,E1 -25682.507,E2 -25682.507} C_VEL
LIN {X 0,Y 133.001,Z 497.513,A -85,B 0,C 180,E1 -25684.034,E2 -25684.034} C_VEL
LIN {X 0,Y 133.017,Z 489.764,A -85,B 0,C 180,E1 -25686.679,E2 -25686.679} C_VEL
LIN {X 0,Y 132.927,Z 481.594,A -85,B 0,C 180,E1 -25689.124,E2 -25689.124} C_VEL
LIN {X 0,Y 133.738,Z 476.295,A -85,B 0,C 180,E1 -25690.286,E2 -25690.286} C_VEL
LIN {X 0,Y 136.47,Z 464.671,A -85,B 0,C 180,E1 -25692.03,E2 -25692.03} C_VEL
LIN {X 0,Y 138.717,Z 451.488,A -85,B 0,C 180,E1 -25693.407,E2 -25693.407} C_VEL
LIN {X 0,Y 140.158,Z 438.999,A -85,B 0,C 180,E1 -25694.205,E2 -25694.205} C_VEL
LIN {X 0,Y 142.698,Z 398.489,A -85,B 0,C 180,E1 -25696.023,E2 -25696.023} C_VEL
LIN {X 0,Y 142.119,Z 391.544,A -85,B 0,C 180,E1 -25696.674,E2 -25696.674} C_VEL
